FUNCTION_BLOCK "Sq_Process_IndexingUnit01"   // FB2111, GRAPH_PLUS
{ S7_Optimized_Access := 'TRUE' }
VERSION : 0.1
   VAR_INPUT
      OFF_SQ : Bool := false;   // Kette ausschalten
      INIT_SQ : Bool := false;   // Kette in Initialzustand versetzen
      ACK_EF : Bool := false;   // Alle Fehler und Störungen quittieren
      S_PREV : Bool := false;   // Vorherigen Schritt am Parameter S_NO ausgeben
      S_NEXT : Bool := false;   // Nächsten Schritt am Parameter S_NO anzeigen
      SW_AUTO : Bool := false;   // Automatischer Betrieb
      SW_TAP : Bool := false;   // Halbautomatisch/Weiterschalten mit Transition
      SW_TOP : Bool := false;   // Halbautomatisch/Ignoriere Transition
      SW_MAN : Bool := false;   // Handbetrieb
      S_SEL : Int := 0;   // Schritt auswählen, der an S_NO ausgegeben werden soll
      S_ON : Bool := false;   // Schritt aktivieren, der an Parameter S_NO anliegt
      S_OFF : Bool := false;   // Schritt deaktivieren, der an Parameter S_NO anliegt
      T_PUSH : Bool := false;   // Schaltfreigabe für Transition im halbautomatischen Betrieb
      ixStart : Bool := true;   // Startfreigabe
      ixCarrierPresent : Bool;   // WT auf dem Indexer vorhanden
      ixCheckTargetReached : Bool := false;   // 0 = Keine Sensor-Zielüberwachung nach Lift vorhanden
      ixTargetReached : Bool := false;   // WT-Sensor des nächsten Ziels
      ixReleaseHoming : Bool;   // Freigabe Grundstellungsfahrt
      ixReleaseTransfer : Bool := true;   // Freigabe der nächsten Position um WT weiterzutakten
      itCarrierReactionDelay : Time := T#350ms;   // Verzögerungszeit für die WT-Erkennung
      itMaxRuntime : Time := t#10s;   // Maximale Laufzeit für diesen Prozess
   END_VAR
   VAR_OUTPUT
      S_NO : Int := 0;   // Schrittnummer
      S_MORE : Bool := false;   // Weitere Schritte sind vorhanden und können in S_NO angezeigt werden.
      S_ACTIVE : Bool := false;   // Schritt, der an Parameter S_NO angezeigt wird, ist aktiv
      ERR_FLT : Bool := false;   // Sammelfehler Interlock oder Supervision
      AUTO_ON : Bool := false;   // Automatischer Betrieb eingeschaltet
      TAP_ON : Bool := false;   // Halbautomatischer Betrieb/Schritt mit Transition eingeschaltet
      TOP_ON : Bool := false;   // Halbautomatischer Betrieb/Ignoriere Transition eingeschaltet
      MAN_ON : Bool := false;   // Handbetrieb eingeschaltet
      qxIsActive : Bool;   // Schrittkette läuft
      qxIsInHome : Bool;   // steht in Grundstellung
      qxCarrierIsDone : Bool;   // WT-Träger ist fertig bearbeitet worden
   END_VAR
   VAR_IN_OUT
      signals : "typeStationSignals";   // Stationssteuersignale
      sq : "typeStepSequence";   // Schrittkettensteuersignale
      cylinder_lift : "typeActor_2Out2In";   // Aktor des Heber
      cylinder_stopper : "typeActor_1Out1In";   // Aktor für den Stopper
      releaseWorkStep : Bool;   // Freigabe für den externen Arbeitsschritt (muss extern zurückgesetzt werden)
   END_VAR
   VAR
      sstReleaseCycle : Struct
         ErrorAck : Bool;
         No_LastCycle : Int;
         T : Time;   // Aktive Zeit des ReleaseCycle
         Tck : Time;
         TckPrev : Time;
      END_STRUCT;
      sinstCarrierOnIndexer : TON_TIME;
      sinstCarrierLeftIndexer : TON_TIME;
      HMI_INFO : Array[0..8] of UInt;
      IF_PAR : G7_IfParPlus_V6;
      RT_DATA : G7_RTDataPlus_V6;   // Interner Datenbereich
      Automatikablauf : G7_TransitionPlus_V6;   // Transitionsstruktur
      Freigabe : G7_TransitionPlus_V6;   // Transitionsstruktur
      Trans3 : G7_TransitionPlus_V6;   // Transitionsstruktur
      Fertig : G7_TransitionPlus_V6;   // Transitionsstruktur
      Grundstellungsfahrt : G7_TransitionPlus_V6;   // Transitionsstruktur
      GST_Aktiv : G7_TransitionPlus_V6;   // Transitionsstruktur
      GST_Beendet : G7_TransitionPlus_V6;   // Transitionsstruktur
      Beendet : G7_TransitionPlus_V6;   // Transitionsstruktur
      TargetIsReached : G7_TransitionPlus_V6;   // Transitionsstruktur / Transition structure
      "Lift steht in Grundstellung_1" : G7_TransitionPlus_V6;   // Transitionsstruktur / Transition structure
      "Lift steht in Arbeitsstellung_1" : G7_TransitionPlus_V6;   // Transitionsstruktur / Transition structure
      "Lift steht in Arbeitsstellung_2" : G7_TransitionPlus_V6;   // Transitionsstruktur / Transition structure
      "WT hat Stopper verlassen" : G7_TransitionPlus_V6;   // Transitionsstruktur / Transition structure
      CarrierIsNotDone : G7_TransitionPlus_V6;   // Transitionsstruktur / Transition structure
      CarrierIsDone : G7_TransitionPlus_V6;   // Transitionsstruktur / Transition structure
      WorkstepDone : G7_TransitionPlus_V6;   // Transitionsstruktur / Transition structure
      NotDone : G7_TransitionPlus_V6;   // Transitionsstruktur / Transition structure
      WorkstepIsReleased : G7_TransitionPlus_V6;   // Transitionsstruktur / Transition structure
      EndzielFrei : G7_TransitionPlus_V6;   // Transitionsstruktur / Transition structure
      EndzielNichtFrei : G7_TransitionPlus_V6;   // Transitionsstruktur / Transition structure
      JogT2 : G7_TransitionPlus_V6;   // Transitionsstruktur / Transition structure
      JogT4 : G7_TransitionPlus_V6;   // Transitionsstruktur / Transition structure
      JogT1 : G7_TransitionPlus_V6;   // Transitionsstruktur / Transition structure
      GatesClosed : G7_TransitionPlus_V6;   // Transitionsstruktur / Transition structure
      GatesOpened : G7_TransitionPlus_V6;   // Transitionsstruktur / Transition structure
      JogT3 : G7_TransitionPlus_V6;   // Transitionsstruktur / Transition structure
      GS_GatesOpened : G7_TransitionPlus_V6;   // Transitionsstruktur / Transition structure
      Initialschritt : G7_StepPlus_V6;   // Schrittstruktur
      Grundstellung : G7_StepPlus_V6;   // Schrittstruktur
      SK_läuft : G7_StepPlus_V6;   // Schrittstruktur
      Fertigmeldung : G7_StepPlus_V6;   // Schrittstruktur
      "Start Grundstellungsfahrt" : G7_StepPlus_V6;   // Schrittstruktur
      "Fertig Grundstellungsfahrt" : G7_StepPlus_V6;   // Schrittstruktur
      Ende : G7_StepPlus_V6;   // Schrittstruktur
      WaitForTarget : G7_StepPlus_V6;   // Schrittstruktur / Step structure
      GS_CylHome : G7_StepPlus_V6;   // Schrittstruktur / Step structure
      IndexerWorkPos : G7_StepPlus_V6;   // Schrittstruktur / Step structure
      IndexerHomePos : G7_StepPlus_V6;   // Schrittstruktur / Step structure
      OpenStopper : G7_StepPlus_V6;   // Schrittstruktur / Step structure
      Decision : G7_StepPlus_V6;   // Schrittstruktur / Step structure
      CheckWorkstepDone : G7_StepPlus_V6;   // Schrittstruktur / Step structure
      Release : G7_StepPlus_V6;   // Schrittstruktur / Step structure
      Warte_Endziel_frei : G7_StepPlus_V6;   // Schrittstruktur / Step structure
      JogS2 : G7_StepPlus_V6;   // Schrittstruktur / Step structure
      JogS4 : G7_StepPlus_V6;   // Schrittstruktur / Step structure
      JogS1 : G7_StepPlus_V6;   // Schrittstruktur / Step structure
      CloseGates : G7_StepPlus_V6;   // Schrittstruktur / Step structure
      OpenGates : G7_StepPlus_V6;   // Schrittstruktur / Step structure
      JogS3 : G7_StepPlus_V6;   // Schrittstruktur / Step structure
      GS_OpenGates : G7_StepPlus_V6;   // Schrittstruktur / Step structure
      SINI : Array[0..1] of USInt;
      LSTT : Array[0..26] of USInt;
      ATAJ : Array[0..26] of USInt;
      ATAB : Array[0..26] of USInt;
      PSTT : Array[0..26] of USInt;
      NSTT : Array[0..26] of USInt;
      ASSJ : Array[0..22] of USInt;
      ASSB : Array[0..22] of USInt;
      PTTS : Array[0..22] of USInt;
      NTTS : Array[0..22] of USInt;
      SW_SQTS : Array[0..22] of USInt;
      SWITCH : Array[0..7] of USInt;
      TVX : Array[0..9] of USInt;
      TTX : Array[0..9] of USInt;
      TSX : Array[0..1] of USInt;
      S00X : Array[0..1] of USInt;
      SOFFX : Array[0..1] of USInt;
      SONX : Array[0..1] of USInt;
      SAX : Array[0..1] of USInt;
      SERRX : Array[0..23] of USInt;
      SMX : Array[0..23] of USInt;
      S0X : Array[0..23] of USInt;
      S1X : Array[0..23] of USInt;
      IL_ALARM_INST : Diag_Alarm;
      SUP_ALARM_INST : Diag_Alarm;
      STEP_TIME_ALARM_INST : Diag_Alarm;
      IEC_TIMER_INST : IEC_TIMER;
      TRANSACTION_FLAG : Bool := false;
   END_VAR
   VAR_TEMP
      txStartCondition : Bool;
      tdTckDiff : DInt;
      txCheckWorkStep : Bool;
   END_VAR
   VAR_TEMP   // added for the SCL form of the ladder/FBD networks
      _w1 : Bool;
      _w2 : Bool;
   END_VAR
   // SINI[0] := 2;
   // LSTT[0] := 255;
   // LSTT[1] := 255;
   // LSTT[2] := 255;
   // LSTT[3] := 255;
   // LSTT[4] := 255;
   // LSTT[5] := 255;
   // LSTT[6] := 255;
   // LSTT[7] := 1;
   // ATAJ[1] := 1;
   // ATAJ[2] := 2;
   // ATAJ[3] := 6;
   // ATAJ[4] := 4;
   // ATAJ[5] := 5;
   // ATAJ[6] := 3;
   // ATAJ[7] := 7;
   // ATAB[0] := 4;
   // ATAB[1] := 1;
   // ATAB[2] := 2;
   // ATAB[3] := 3;
   // ATAB[5] := 5;
   // ATAB[6] := 6;
   // ATAB[7] := 7;
   // PSTT[1] := 1;
   // PSTT[2] := 2;
   // PSTT[3] := 3;
   // PSTT[5] := 4;
   // PSTT[6] := 5;
   // PSTT[7] := 6;
   // NSTT[0] := 1;
   // NSTT[1] := 2;
   // NSTT[2] := 12;
   // NSTT[3] := 6;
   // NSTT[4] := 4;
   // NSTT[5] := 8;
   // NSTT[6] := 6;
   // NSTT[7] := 1;
   // ASSJ[1] := 1;
   // ASSJ[2] := 2;
   // ASSJ[3] := 3;
   // ASSJ[4] := 4;
   // ASSJ[5] := 5;
   // ASSJ[6] := 6;
   // ASSB[1] := 1;
   // ASSB[2] := 2;
   // ASSB[3] := 3;
   // ASSB[4] := 4;
   // ASSB[5] := 5;
   // ASSB[6] := 6;
   // PTTS[0] := 255;
   // PTTS[2] := 1;
   // PTTS[3] := 8;
   // PTTS[4] := 4;
   // PTTS[5] := 26;
   // PTTS[6] := 3;
   // NTTS[1] := 1;
   // NTTS[2] := 2;
   // NTTS[3] := 3;
   // NTTS[4] := 5;
   // NTTS[5] := 6;
   // NTTS[6] := 7;
   // SW_SQTS[1] := 1;
   // SW_SQTS[2] := 1;
   // SW_SQTS[3] := 2;
   // SW_SQTS[4] := 3;
   // SW_SQTS[5] := 3;
   // SW_SQTS[6] := 4;
   // TVX[0] := 16#1;
   // TTX[0] := 16#1;
   // TSX[0] := 16#1;
   // S00X[0] := 16#1;
   // SOFFX[0] := 16#1;
   // SONX[0] := 16#1;
   // SAX[0] := 16#1;
   // SERRX[0] := 16#1;
   // SMX[0] := 16#1;
   // S0X[0] := 16#1;
   // S1X[0] := 16#1;
   // LSTT[8] := 255;
   // ATAJ[8] := 8;
   // ATAB[8] := 8;
   // PSTT[8] := 7;
   // NSTT[8] := 3;
   // ASSJ[7] := 7;
   // ASSB[7] := 7;
   // PTTS[7] := 12;
   // NTTS[7] := 8;
   // SW_SQTS[7] := 2;
   // LSTT[9] := 255;
   // LSTT[10] := 255;
   // LSTT[11] := 255;
   // ATAJ[9] := 9;
   // ATAJ[10] := 10;
   // ATAJ[11] := 14;
   // ATAB[9] := 9;
   // ATAB[10] := 10;
   // ATAB[11] := 11;
   // PSTT[9] := 8;
   // PSTT[10] := 9;
   // PSTT[11] := 10;
   // NSTT[9] := 22;
   // NSTT[10] := 18;
   // NSTT[11] := 17;
   // ASSJ[8] := 8;
   // ASSJ[9] := 9;
   // ASSJ[10] := 10;
   // ASSB[8] := 8;
   // ASSB[9] := 9;
   // ASSB[10] := 10;
   // PTTS[8] := 5;
   // PTTS[9] := 13;
   // PTTS[10] := 25;
   // NTTS[8] := 9;
   // NTTS[9] := 10;
   // NTTS[10] := 11;
   // SW_SQTS[8] := 3;
   // SW_SQTS[9] := 5;
   // SW_SQTS[10] := 6;
   // LSTT[12] := 255;
   // LSTT[13] := 255;
   // ATAJ[12] := 12;
   // ATAJ[13] := 13;
   // ATAB[12] := 12;
   // ATAB[13] := 14;
   // PSTT[12] := 11;
   // PSTT[13] := 12;
   // NSTT[12] := 7;
   // NSTT[13] := 9;
   // ASSJ[11] := 11;
   // ASSJ[12] := 12;
   // ASSB[11] := 11;
   // ASSB[12] := 12;
   // PTTS[11] := 18;
   // PTTS[12] := 2;
   // NTTS[11] := 12;
   // NTTS[12] := 13;
   // SW_SQTS[11] := 2;
   // SW_SQTS[12] := 1;
   // LSTT[14] := 255;
   // LSTT[15] := 255;
   // ATAJ[14] := 11;
   // ATAJ[15] := 15;
   // ATAB[14] := 13;
   // ATAB[15] := 16;
   // PSTT[14] := 12;
   // PSTT[15] := 13;
   // NSTT[14] := 17;
   // NSTT[15] := 20;
   // ASSJ[13] := 13;
   // ASSJ[14] := 14;
   // ASSB[13] := 13;
   // ASSB[14] := 14;
   // PTTS[13] := 20;
   // PTTS[14] := 23;
   // NTTS[13] := 15;
   // NTTS[14] := 17;
   // SW_SQTS[13] := 5;
   // SW_SQTS[14] := 5;
   // LSTT[16] := 16;
   // ATAJ[16] := 16;
   // ATAB[16] := 15;
   // PSTT[16] := 13;
   // NSTT[16] := 16;
   // LSTT[17] := 255;
   // LSTT[18] := 255;
   // ATAJ[17] := 17;
   // ATAJ[18] := 18;
   // ATAB[17] := 17;
   // ATAB[18] := 19;
   // PSTT[17] := 14;
   // PSTT[18] := 15;
   // NSTT[17] := 16;
   // NSTT[18] := 11;
   // ASSJ[15] := 15;
   // ASSB[15] := 15;
   // PTTS[15] := 21;
   // NTTS[15] := 18;
   // SW_SQTS[15] := 7;
   // LSTT[19] := 17;
   // ATAJ[19] := 19;
   // ATAB[19] := 18;
   // PSTT[19] := 15;
   // NSTT[19] := 17;
   // ASSJ[16] := 16;
   // ASSB[16] := 16;
   // PTTS[16] := 17;
   // NTTS[16] := 20;
   // SW_SQTS[16] := 5;
   // LSTT[20] := 255;
   // LSTT[21] := 255;
   // LSTT[22] := 255;
   // LSTT[23] := 255;
   // LSTT[24] := 255;
   // LSTT[25] := 255;
   // ATAJ[20] := 20;
   // ATAJ[21] := 21;
   // ATAJ[22] := 22;
   // ATAJ[23] := 23;
   // ATAJ[24] := 24;
   // ATAJ[25] := 25;
   // ATAB[20] := 20;
   // ATAB[21] := 21;
   // ATAB[22] := 22;
   // ATAB[23] := 23;
   // ATAB[24] := 24;
   // ATAB[25] := 25;
   // PSTT[20] := 16;
   // PSTT[21] := 17;
   // PSTT[22] := 18;
   // PSTT[23] := 19;
   // PSTT[24] := 20;
   // PSTT[25] := 21;
   // NSTT[20] := 13;
   // NSTT[21] := 15;
   // NSTT[22] := 19;
   // NSTT[23] := 14;
   // NSTT[24] := 21;
   // NSTT[25] := 10;
   // ASSJ[17] := 17;
   // ASSJ[18] := 18;
   // ASSJ[19] := 19;
   // ASSJ[20] := 20;
   // ASSJ[21] := 21;
   // ASSB[17] := 17;
   // ASSB[18] := 18;
   // ASSB[19] := 19;
   // ASSB[20] := 20;
   // ASSB[21] := 21;
   // PTTS[17] := 11;
   // PTTS[18] := 10;
   // PTTS[19] := 22;
   // PTTS[20] := 15;
   // PTTS[21] := 24;
   // NTTS[17] := 21;
   // NTTS[18] := 22;
   // NTTS[19] := 23;
   // NTTS[20] := 24;
   // NTTS[21] := 25;
   // SW_SQTS[17] := 7;
   // SW_SQTS[18] := 5;
   // SW_SQTS[19] := 5;
   // SW_SQTS[20] := 6;
   // SW_SQTS[21] := 6;
   // LSTT[26] := 255;
   // ATAJ[26] := 26;
   // ATAB[26] := 26;
   // PSTT[26] := 22;
   // NSTT[26] := 5;
   // ASSJ[22] := 22;
   // ASSB[22] := 22;
   // PTTS[22] := 9;
   // NTTS[22] := 26;
   // SW_SQTS[22] := 3;
BEGIN
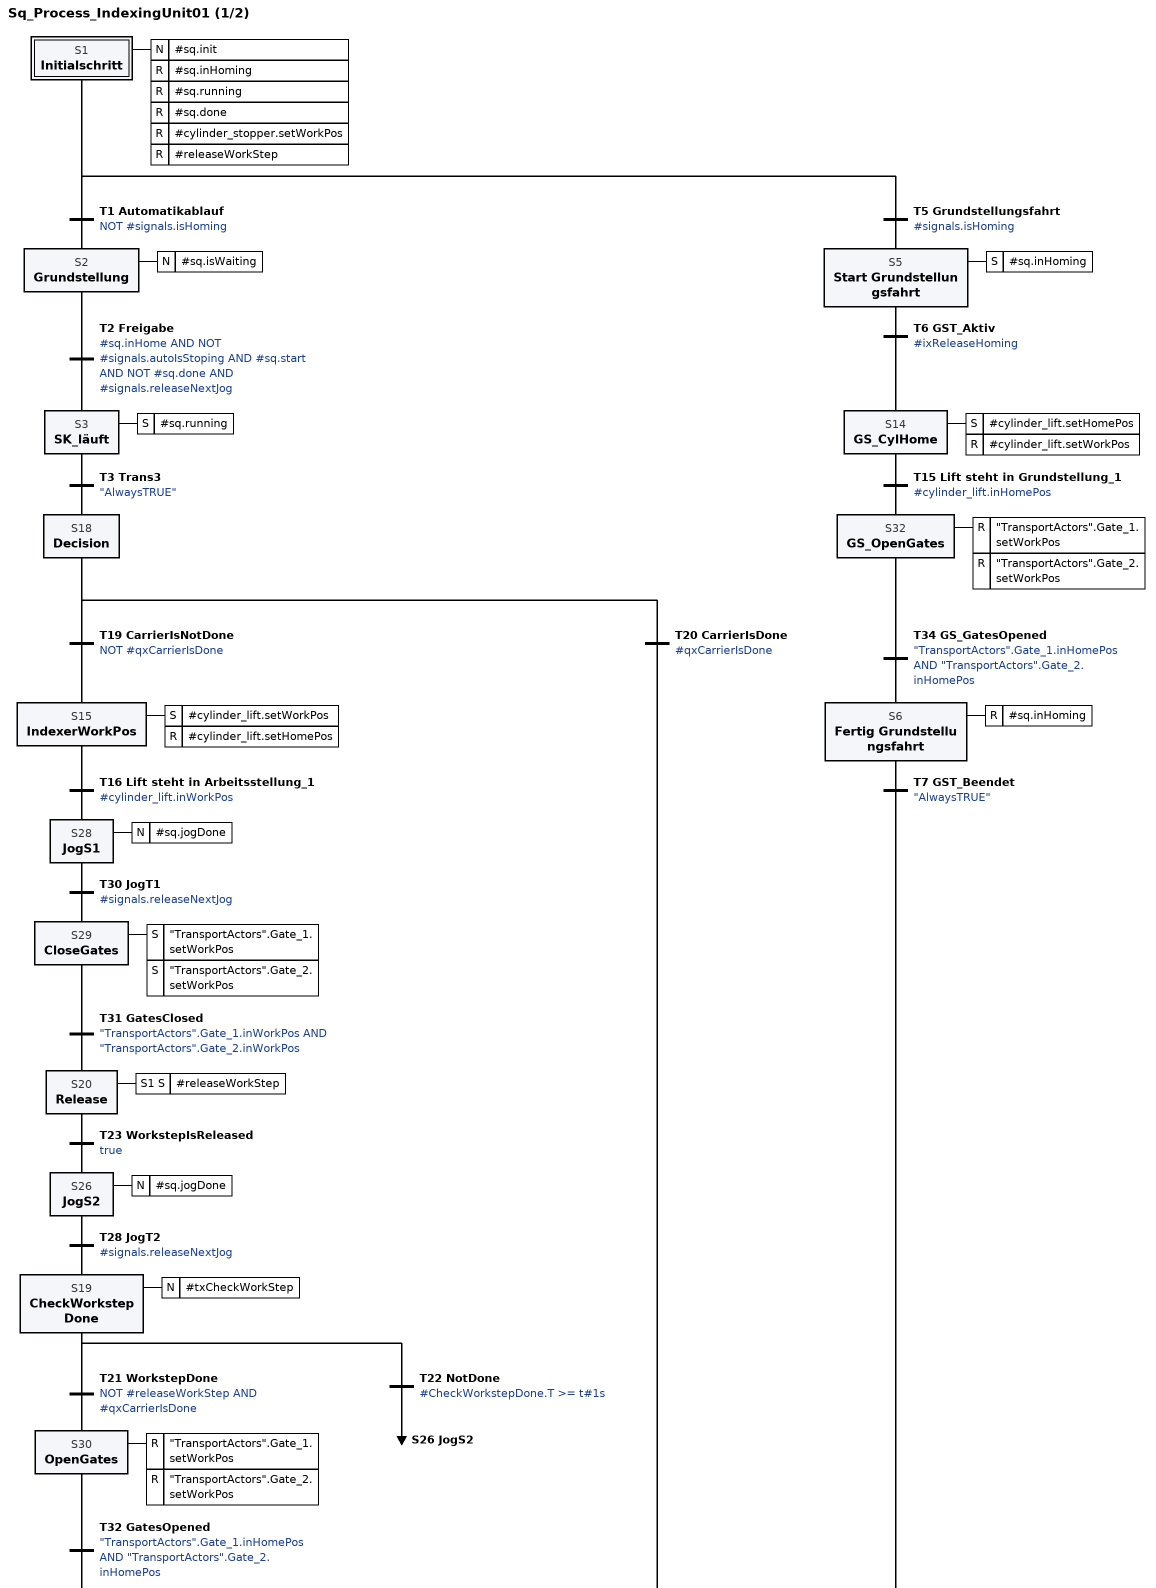
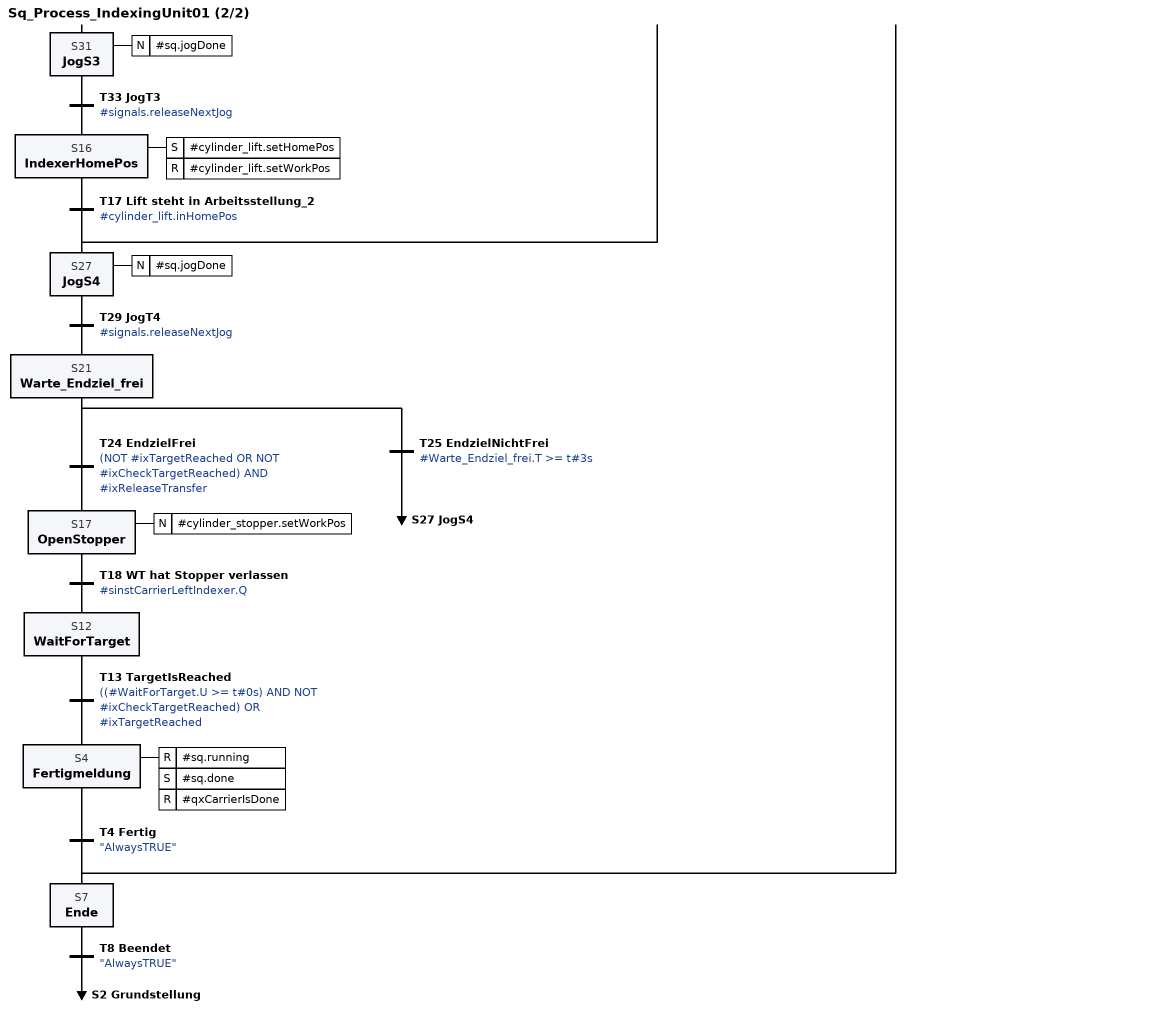
   // permanent pre-instructions
   NETWORK 1
   TITLE = Schrittkette verfügbar
      #sq.exists := true;
   NETWORK 2
   TITLE = WT auf dem Indexer
      #sinstCarrierOnIndexer(IN := #ixCarrierPresent, PT := #itCarrierReactionDelay);   // TON
   NETWORK 3
   TITLE = WT hat den Indexer verlassen
      #sinstCarrierLeftIndexer(IN := NOT #ixCarrierPresent, PT := #itCarrierReactionDelay);   // TON
   NETWORK 4
   TITLE = Schrittkette in Grundstellung (Erweitern)
      #sq.inHome := #Grundstellung.X AND #cylinder_lift.inHomePos AND #cylinder_stopper.inHomePos AND "TransportActors".Gate_1.inHomePos AND "TransportActors".Gate_2.inHomePos;
   NETWORK 5
   TITLE = Startbedingung (Erweitern)
      #txStartCondition := #ixStart AND #sinstCarrierOnIndexer.Q;
   NETWORK 6
   TITLE = Schrittkette starten
      #sq.start := #sq.inHome AND NOT #sq.running AND #signals.releaseCycle AND NOT #signals.isHoming AND #txStartCondition;
      IF #sq.start THEN #sq.done := FALSE; END_IF;
   NETWORK 7
   TITLE = ReleaseCycle Timer
      // ENO of a box is taken as its EN; it also drops when the box reports an error
      #_w1 := #ERR_FLT AND #ACK_EF;
      #_w2 := #_w1 AND NOT #sstReleaseCycle.ErrorAck;   // rising edge
      #sstReleaseCycle.ErrorAck := #_w1;
      IF (#S_NO <> #sstReleaseCycle.No_LastCycle) OR #_w2 THEN
          #sstReleaseCycle.T := T#0MS;
          #sstReleaseCycle.TckPrev := #sstReleaseCycle.Tck;
          #sstReleaseCycle.No_LastCycle := #S_NO;
      END_IF;
      #sstReleaseCycle.Tck := TIME_TCK();
      #tdTckDiff := #sstReleaseCycle.Tck - #sstReleaseCycle.TckPrev;
      #sstReleaseCycle.TckPrev := #sstReleaseCycle.Tck;
      IF (0 <= #tdTckDiff) AND (#tdTckDiff <= 1000) AND #signals.releaseCycle THEN
          #sstReleaseCycle.T := #sstReleaseCycle.T + #tdTckDiff;
      END_IF;

   // sequencer 1
   INITIAL_STEP Initialschritt:   // S1, max time T#10S, warning time T#7S
              N    #sq.init
              R    #sq.inHoming
              R    #sq.running
              R    #sq.done
              R    #cylinder_stopper.setWorkPos
              R    #releaseWorkStep
   END_STEP
   TRANSITION Automatikablauf FROM Initialschritt TO Grundstellung   // T1
      := NOT #signals.isHoming;
   END_TRANSITION
   TRANSITION Grundstellungsfahrt FROM Initialschritt TO "Start Grundstellungsfahrt"   // T5
      := #signals.isHoming;
   END_TRANSITION
   STEP Grundstellung:   // S2, max time T#10S, warning time T#7S
              N    #sq.isWaiting
   END_STEP
   TRANSITION Freigabe FROM Grundstellung TO SK_läuft   // T2
      := #sq.inHome AND NOT #signals.autoIsStoping AND #sq.start AND NOT #sq.done AND #signals.releaseNextJog;
   END_TRANSITION
   STEP SK_läuft:   // S3, max time T#10S, warning time T#7S
              S    #sq.running
   END_STEP
   TRANSITION Trans3 FROM SK_läuft TO Decision   // T3
      := "AlwaysTRUE";
   END_TRANSITION
   STEP Fertigmeldung:   // S4, max time T#10S, warning time T#7S
              R    #sq.running
              S    #sq.done
              R    #qxCarrierIsDone
   END_STEP
   TRANSITION Fertig FROM Fertigmeldung TO Ende   // T4
      := "AlwaysTRUE";
   END_TRANSITION
   STEP "Start Grundstellungsfahrt":   // S5, max time T#10S, warning time T#7S
              S    #sq.inHoming
   END_STEP
   TRANSITION GST_Aktiv FROM "Start Grundstellungsfahrt" TO GS_CylHome   // T6
      := #ixReleaseHoming;
   END_TRANSITION
   STEP "Fertig Grundstellungsfahrt":   // S6, max time T#10S, warning time T#7S
              R    #sq.inHoming
   END_STEP
   TRANSITION GST_Beendet FROM "Fertig Grundstellungsfahrt" TO Ende   // T7
      := "AlwaysTRUE";
   END_TRANSITION
   STEP Ende:   // S7, max time T#10S, warning time T#7S
   END_STEP
   TRANSITION Beendet FROM Ende TO Grundstellung   // T8, jump
      := "AlwaysTRUE";
   END_TRANSITION
   STEP JogS2:   // S26, max time T#10S, warning time T#7S
              N    #sq.jogDone
   END_STEP
   TRANSITION JogT2 FROM JogS2 TO CheckWorkstepDone   // T28
      := #signals.releaseNextJog;
   END_TRANSITION
   STEP IndexerHomePos:   // S16, max time T#10S, warning time T#7S
      supervision V := #IndexerHomePos.X AND #cylinder_lift.inError;
              S    #cylinder_lift.setHomePos
              R    #cylinder_lift.setWorkPos
   END_STEP
   TRANSITION "Lift steht in Arbeitsstellung_2" FROM IndexerHomePos TO JogS4   // T17
      := #cylinder_lift.inHomePos;
   END_TRANSITION
   STEP OpenStopper:   // S17, max time T#10S, warning time T#7S
      supervision V := #OpenStopper.X AND #cylinder_stopper.inError;
              N    #cylinder_stopper.setWorkPos
   END_STEP
   TRANSITION "WT hat Stopper verlassen" FROM OpenStopper TO WaitForTarget   // T18
      := #sinstCarrierLeftIndexer.Q;
   END_TRANSITION
   STEP JogS4:   // S27, max time T#10S, warning time T#7S
              N    #sq.jogDone
   END_STEP
   TRANSITION JogT4 FROM JogS4 TO Warte_Endziel_frei   // T29
      := #signals.releaseNextJog;
   END_TRANSITION
   STEP WaitForTarget:   // S12, max time T#10S, warning time T#7S
      supervision V := #sstReleaseCycle.T >= #itMaxRuntime;
   END_STEP
   TRANSITION TargetIsReached FROM WaitForTarget TO Fertigmeldung   // T13
      := ((#WaitForTarget.U >= t#0s) AND NOT #ixCheckTargetReached) OR #ixTargetReached;
   END_TRANSITION
   STEP Decision:   // S18, max time T#10S, warning time T#7S
   END_STEP
   TRANSITION CarrierIsNotDone FROM Decision TO IndexerWorkPos   // T19
      := NOT #qxCarrierIsDone;
   END_TRANSITION
   TRANSITION CarrierIsDone FROM Decision TO JogS4   // T20
      := #qxCarrierIsDone;
   END_TRANSITION
   STEP GS_CylHome:   // S14, max time T#10S, warning time T#7S
      supervision V := #GS_CylHome.X AND #cylinder_lift.inError;
              S    #cylinder_lift.setHomePos
              R    #cylinder_lift.setWorkPos
   END_STEP
   TRANSITION "Lift steht in Grundstellung_1" FROM GS_CylHome TO GS_OpenGates   // T15
      := #cylinder_lift.inHomePos;
   END_TRANSITION
   STEP IndexerWorkPos:   // S15, max time T#10S, warning time T#7S
      supervision V := #IndexerWorkPos.X AND #cylinder_lift.inError;
              S    #cylinder_lift.setWorkPos
              R    #cylinder_lift.setHomePos
   END_STEP
   TRANSITION "Lift steht in Arbeitsstellung_1" FROM IndexerWorkPos TO JogS1   // T16
      := #cylinder_lift.inWorkPos;
   END_TRANSITION
   STEP CheckWorkstepDone:   // S19, max time T#10S, warning time T#7S
              N    #txCheckWorkStep
   END_STEP
   TRANSITION WorkstepDone FROM CheckWorkstepDone TO OpenGates   // T21
      := NOT #releaseWorkStep AND #qxCarrierIsDone;
   END_TRANSITION
   TRANSITION NotDone FROM CheckWorkstepDone TO JogS2   // T22, jump
      := #CheckWorkstepDone.T >= t#1s;
   END_TRANSITION
   STEP Release:   // S20, max time T#10S, warning time T#7S
          S1  S    #releaseWorkStep
   END_STEP
   TRANSITION WorkstepIsReleased FROM Release TO JogS2   // T23
      := true;
   END_TRANSITION
   STEP Warte_Endziel_frei:   // S21, max time T#10S, warning time T#7S
   END_STEP
   TRANSITION EndzielFrei FROM Warte_Endziel_frei TO OpenStopper   // T24
      := (NOT #ixTargetReached OR NOT #ixCheckTargetReached) AND #ixReleaseTransfer;
   END_TRANSITION
   TRANSITION EndzielNichtFrei FROM Warte_Endziel_frei TO JogS4   // T25, jump
      := #Warte_Endziel_frei.T >= t#3s;
   END_TRANSITION
   STEP JogS1:   // S28, max time T#10S, warning time T#7S
              N    #sq.jogDone
   END_STEP
   TRANSITION JogT1 FROM JogS1 TO CloseGates   // T30
      := #signals.releaseNextJog;
   END_TRANSITION
   STEP CloseGates:   // S29, max time T#10S, warning time T#7S
      supervision V := (#sstReleaseCycle.T >= #itMaxRuntime) OR (("TransportActors".Gate_1.inError OR "TransportActors".Gate_2.inError) AND #CloseGates.X);
              S    "TransportActors".Gate_1.setWorkPos
              S    "TransportActors".Gate_2.setWorkPos
   END_STEP
   TRANSITION GatesClosed FROM CloseGates TO Release   // T31
      := "TransportActors".Gate_1.inWorkPos AND "TransportActors".Gate_2.inWorkPos;
   END_TRANSITION
   STEP OpenGates:   // S30, max time T#10S, warning time T#7S
      supervision V := (#sstReleaseCycle.T >= #itMaxRuntime) OR (("TransportActors".Gate_1.inError OR "TransportActors".Gate_2.inError) AND #OpenGates.X);
              R    "TransportActors".Gate_1.setWorkPos
              R    "TransportActors".Gate_2.setWorkPos
   END_STEP
   TRANSITION GatesOpened FROM OpenGates TO JogS3   // T32
      := "TransportActors".Gate_1.inHomePos AND "TransportActors".Gate_2.inHomePos;
   END_TRANSITION
   STEP JogS3:   // S31, max time T#10S, warning time T#7S
              N    #sq.jogDone
   END_STEP
   TRANSITION JogT3 FROM JogS3 TO IndexerHomePos   // T33
      := #signals.releaseNextJog;
   END_TRANSITION
   STEP GS_OpenGates:   // S32, max time T#10S, warning time T#7S
      supervision V := (#sstReleaseCycle.T >= #itMaxRuntime) OR (("TransportActors".Gate_1.inError OR "TransportActors".Gate_2.inError) AND #GS_OpenGates.X);
              R    "TransportActors".Gate_1.setWorkPos
              R    "TransportActors".Gate_2.setWorkPos
   END_STEP
   TRANSITION GS_GatesOpened FROM GS_OpenGates TO "Fertig Grundstellungsfahrt"   // T34
      := "TransportActors".Gate_1.inHomePos AND "TransportActors".Gate_2.inHomePos;
   END_TRANSITION

   // permanent post-instructions
   NETWORK 1
   TITLE = Störungssignal weitergeben
      #sq.error := #ERR_FLT;
   NETWORK 2
   TITLE = Ablauf ist aktiv
      #qxIsActive := #sq.running;
   NETWORK 3
   TITLE = steht in Grundstellung
      #qxIsInHome := #sq.inHome AND NOT #sq.running;
   NETWORK 4
   TITLE = WT-Träger ist fertig bearbeitet worden
      IF NOT #releaseWorkStep AND #txCheckWorkStep THEN #qxCarrierIsDone := TRUE; END_IF;
END_FUNCTION_BLOCK

FUNCTION "FG10StepSequences" : Void   // FC2010, FBD
TITLE = Schrittkettensteuerung
{ S7_Optimized_Access := 'TRUE' }
VERSION : 0.1
// Ersteller: Andreas Fast Automation
// E-Mail: automation@fast-andreas.de
// 
// Projekt dient zu Demonstrationszwecken und frei genutzt werden.
// 
// Bausteinbeschreibung:
   VAR_IN_OUT
      station : "typeStation";
   END_VAR
   VAR_TEMP
      tempInit : Bool;
      tempAck : Bool;
      tempSwAuto : Bool;
      tempSwMan : Bool;
      tempSwTap : Bool;
      tempPush : Bool;
   END_VAR
BEGIN

REGION Network 1: Graph Parameter
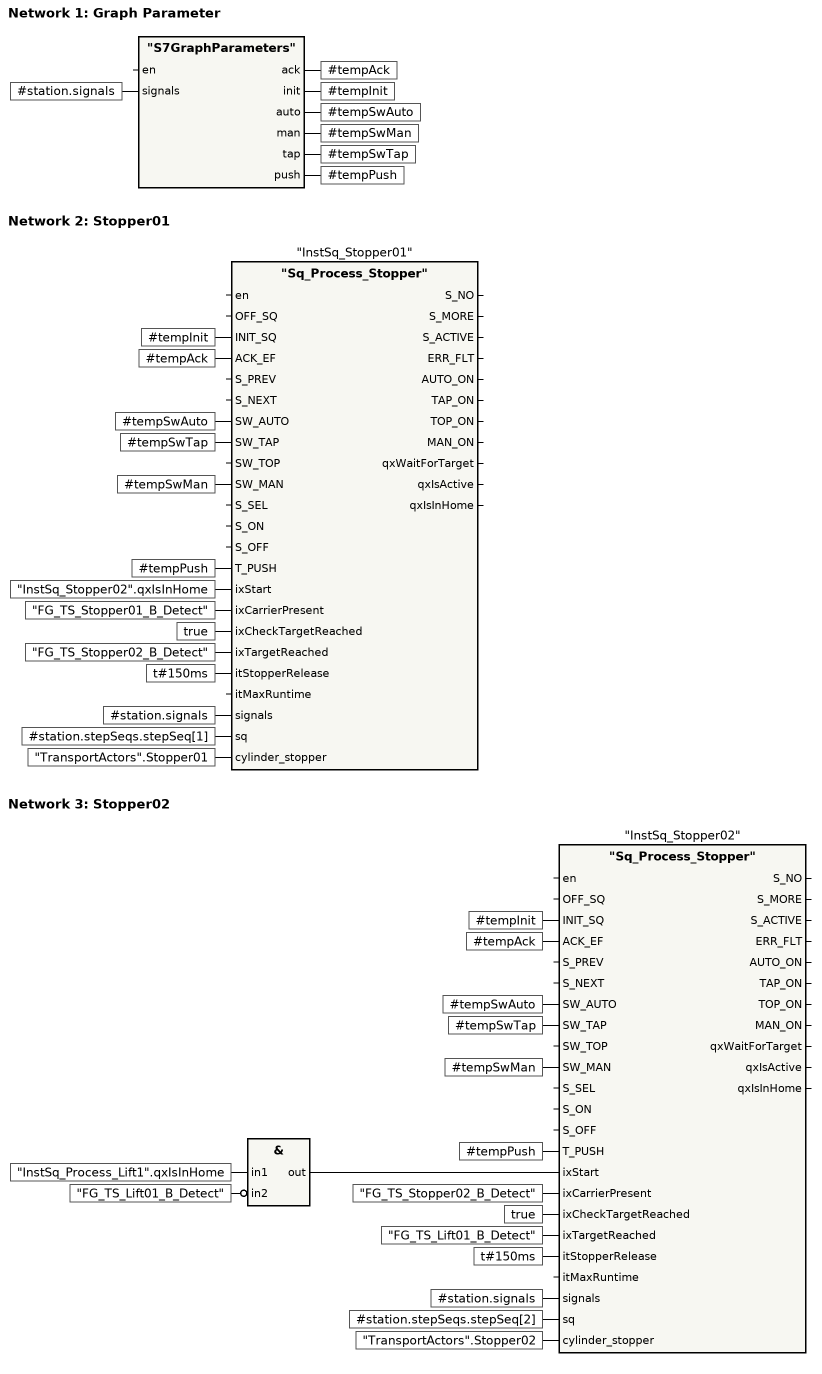
   "S7GraphParameters"(signals := #station.signals,
                       ack => #tempAck,
                       init => #tempInit,
                       auto => #tempSwAuto,
                       man => #tempSwMan,
                       tap => #tempSwTap,
                       push => #tempPush);
END_REGION

REGION Network 2: Stopper01
   "InstSq_Stopper01"(INIT_SQ := #tempInit,   // "Sq_Process_Stopper"
                      ACK_EF := #tempAck,
                      SW_AUTO := #tempSwAuto,
                      SW_TAP := #tempSwTap,
                      SW_MAN := #tempSwMan,
                      T_PUSH := #tempPush,
                      ixStart := "InstSq_Stopper02".qxIsInHome,
                      ixCarrierPresent := "FG_TS_Stopper01_B_Detect",
                      ixCheckTargetReached := true,
                      ixTargetReached := "FG_TS_Stopper02_B_Detect",
                      itStopperRelease := t#150ms,
                      signals := #station.signals,
                      sq := #station.stepSeqs.stepSeq[1],
                      cylinder_stopper := "TransportActors".Stopper01);
END_REGION

REGION Network 3: Stopper02
   "InstSq_Stopper02"(INIT_SQ := #tempInit,   // "Sq_Process_Stopper"
                      ACK_EF := #tempAck,
                      SW_AUTO := #tempSwAuto,
                      SW_TAP := #tempSwTap,
                      SW_MAN := #tempSwMan,
                      T_PUSH := #tempPush,
                      ixStart := "InstSq_Process_Lift1".qxIsInHome AND NOT "FG_TS_Lift01_B_Detect",
                      ixCarrierPresent := "FG_TS_Stopper02_B_Detect",
                      ixCheckTargetReached := true,
                      ixTargetReached := "FG_TS_Lift01_B_Detect",
                      itStopperRelease := t#150ms,
                      signals := #station.signals,
                      sq := #station.stepSeqs.stepSeq[2],
                      cylinder_stopper := "TransportActors".Stopper02);
END_REGION

REGION Network 4: Lift 1
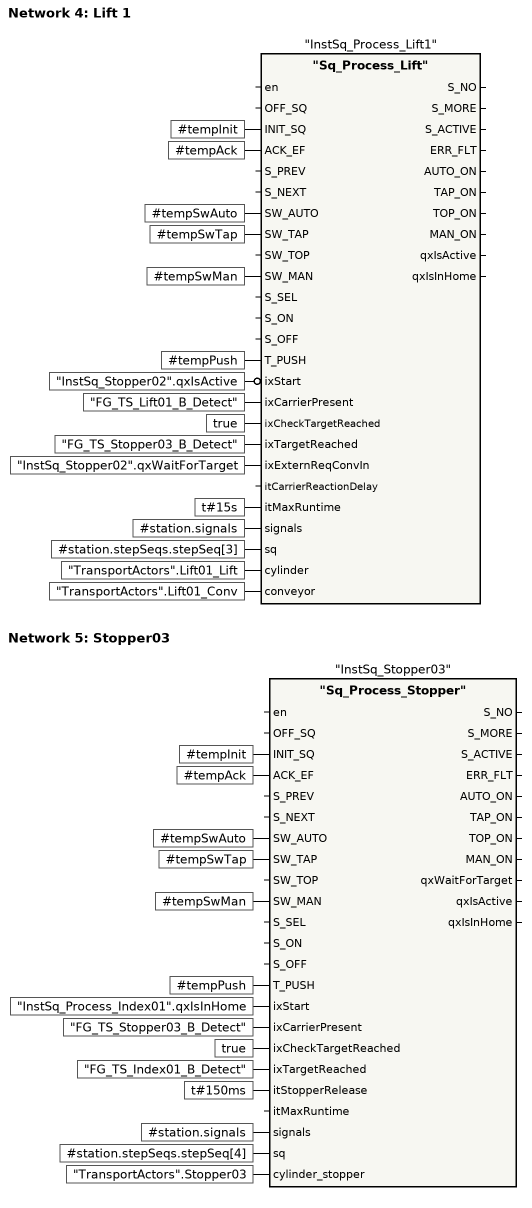
   "InstSq_Process_Lift1"(INIT_SQ := #tempInit,   // "Sq_Process_Lift"
                          ACK_EF := #tempAck,
                          SW_AUTO := #tempSwAuto,
                          SW_TAP := #tempSwTap,
                          SW_MAN := #tempSwMan,
                          T_PUSH := #tempPush,
                          ixStart := NOT "InstSq_Stopper02".qxIsActive,
                          ixCarrierPresent := "FG_TS_Lift01_B_Detect",
                          ixCheckTargetReached := true,
                          ixTargetReached := "FG_TS_Stopper03_B_Detect",
                          ixExternReqConvIn := "InstSq_Stopper02".qxWaitForTarget,
                          itMaxRuntime := t#15s,
                          signals := #station.signals,
                          sq := #station.stepSeqs.stepSeq[3],
                          cylinder := "TransportActors".Lift01_Lift,
                          conveyor := "TransportActors".Lift01_Conv);
END_REGION

REGION Network 5: Stopper03
   "InstSq_Stopper03"(INIT_SQ := #tempInit,   // "Sq_Process_Stopper"
                      ACK_EF := #tempAck,
                      SW_AUTO := #tempSwAuto,
                      SW_TAP := #tempSwTap,
                      SW_MAN := #tempSwMan,
                      T_PUSH := #tempPush,
                      ixStart := "InstSq_Process_Index01".qxIsInHome,
                      ixCarrierPresent := "FG_TS_Stopper03_B_Detect",
                      ixCheckTargetReached := true,
                      ixTargetReached := "FG_TS_Index01_B_Detect",
                      itStopperRelease := t#150ms,
                      signals := #station.signals,
                      sq := #station.stepSeqs.stepSeq[4],
                      cylinder_stopper := "TransportActors".Stopper03);
END_REGION

REGION Network 6: Index01
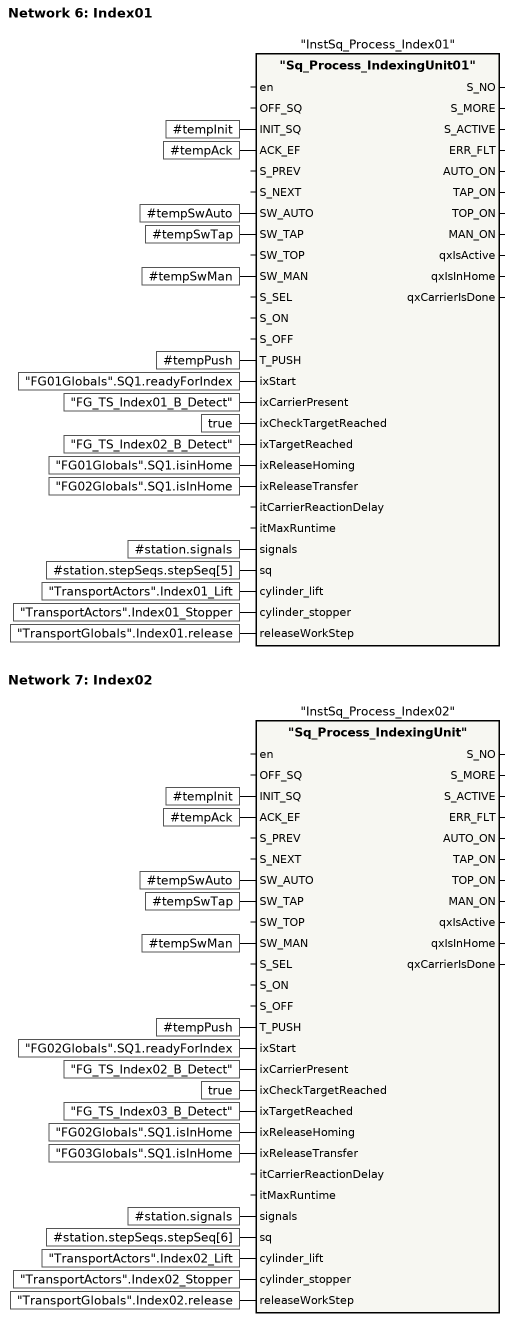
   "InstSq_Process_Index01"(INIT_SQ := #tempInit,   // "Sq_Process_IndexingUnit01"
                           ACK_EF := #tempAck,
                           SW_AUTO := #tempSwAuto,
                           SW_TAP := #tempSwTap,
                           SW_MAN := #tempSwMan,
                           T_PUSH := #tempPush,
                           ixStart := "FG01Globals".SQ1.readyForIndex,
                           ixCarrierPresent := "FG_TS_Index01_B_Detect",
                           ixCheckTargetReached := true,
                           ixTargetReached := "FG_TS_Index02_B_Detect",
                           ixReleaseHoming := "FG01Globals".SQ1.isinHome,
                           ixReleaseTransfer := "FG02Globals".SQ1.isInHome,
                           signals := #station.signals,
                           sq := #station.stepSeqs.stepSeq[5],
                           cylinder_lift := "TransportActors".Index01_Lift,
                           cylinder_stopper := "TransportActors".Index01_Stopper,
                           releaseWorkStep := "TransportGlobals".Index01.release);
END_REGION

REGION Network 7: Index02
   "InstSq_Process_Index02"(INIT_SQ := #tempInit,   // "Sq_Process_IndexingUnit"
                           ACK_EF := #tempAck,
                           SW_AUTO := #tempSwAuto,
                           SW_TAP := #tempSwTap,
                           SW_MAN := #tempSwMan,
                           T_PUSH := #tempPush,
                           ixStart := "FG02Globals".SQ1.readyForIndex,
                           ixCarrierPresent := "FG_TS_Index02_B_Detect",
                           ixCheckTargetReached := true,
                           ixTargetReached := "FG_TS_Index03_B_Detect",
                           ixReleaseHoming := "FG02Globals".SQ1.isInHome,
                           ixReleaseTransfer := "FG03Globals".SQ1.isInHome,
                           signals := #station.signals,
                           sq := #station.stepSeqs.stepSeq[6],
                           cylinder_lift := "TransportActors".Index02_Lift,
                           cylinder_stopper := "TransportActors".Index02_Stopper,
                           releaseWorkStep := "TransportGlobals".Index02.release);
END_REGION

REGION Network 8: Index03
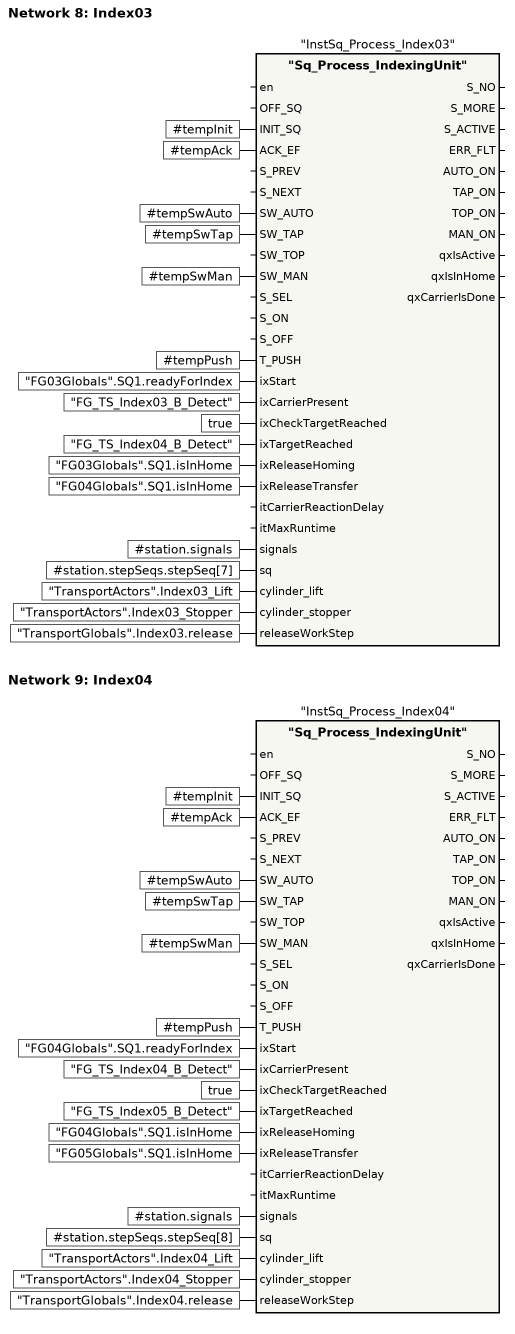
   "InstSq_Process_Index03"(INIT_SQ := #tempInit,   // "Sq_Process_IndexingUnit"
                           ACK_EF := #tempAck,
                           SW_AUTO := #tempSwAuto,
                           SW_TAP := #tempSwTap,
                           SW_MAN := #tempSwMan,
                           T_PUSH := #tempPush,
                           ixStart := "FG03Globals".SQ1.readyForIndex,
                           ixCarrierPresent := "FG_TS_Index03_B_Detect",
                           ixCheckTargetReached := true,
                           ixTargetReached := "FG_TS_Index04_B_Detect",
                           ixReleaseHoming := "FG03Globals".SQ1.isInHome,
                           ixReleaseTransfer := "FG04Globals".SQ1.isInHome,
                           signals := #station.signals,
                           sq := #station.stepSeqs.stepSeq[7],
                           cylinder_lift := "TransportActors".Index03_Lift,
                           cylinder_stopper := "TransportActors".Index03_Stopper,
                           releaseWorkStep := "TransportGlobals".Index03.release);
END_REGION

REGION Network 9: Index04
   "InstSq_Process_Index04"(INIT_SQ := #tempInit,   // "Sq_Process_IndexingUnit"
                           ACK_EF := #tempAck,
                           SW_AUTO := #tempSwAuto,
                           SW_TAP := #tempSwTap,
                           SW_MAN := #tempSwMan,
                           T_PUSH := #tempPush,
                           ixStart := "FG04Globals".SQ1.readyForIndex,
                           ixCarrierPresent := "FG_TS_Index04_B_Detect",
                           ixCheckTargetReached := true,
                           ixTargetReached := "FG_TS_Index05_B_Detect",
                           ixReleaseHoming := "FG04Globals".SQ1.isInHome,
                           ixReleaseTransfer := "FG05Globals".SQ1.isInHome,
                           signals := #station.signals,
                           sq := #station.stepSeqs.stepSeq[8],
                           cylinder_lift := "TransportActors".Index04_Lift,
                           cylinder_stopper := "TransportActors".Index04_Stopper,
                           releaseWorkStep := "TransportGlobals".Index04.release);
END_REGION

REGION Network 10: Index05
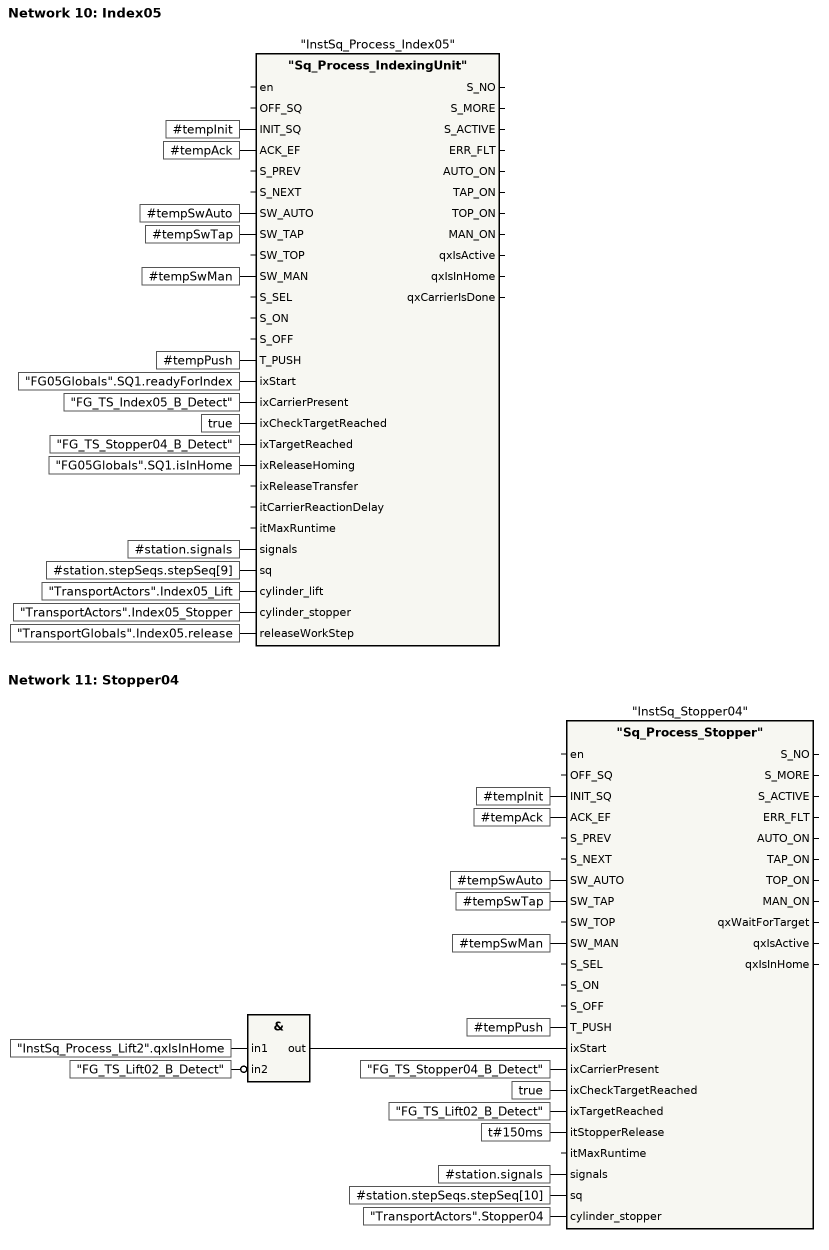
   "InstSq_Process_Index05"(INIT_SQ := #tempInit,   // "Sq_Process_IndexingUnit"
                           ACK_EF := #tempAck,
                           SW_AUTO := #tempSwAuto,
                           SW_TAP := #tempSwTap,
                           SW_MAN := #tempSwMan,
                           T_PUSH := #tempPush,
                           ixStart := "FG05Globals".SQ1.readyForIndex,
                           ixCarrierPresent := "FG_TS_Index05_B_Detect",
                           ixCheckTargetReached := true,
                           ixTargetReached := "FG_TS_Stopper04_B_Detect",
                           ixReleaseHoming := "FG05Globals".SQ1.isInHome,
                           signals := #station.signals,
                           sq := #station.stepSeqs.stepSeq[9],
                           cylinder_lift := "TransportActors".Index05_Lift,
                           cylinder_stopper := "TransportActors".Index05_Stopper,
                           releaseWorkStep := "TransportGlobals".Index05.release);
END_REGION

REGION Network 11: Stopper04
   "InstSq_Stopper04"(INIT_SQ := #tempInit,   // "Sq_Process_Stopper"
                      ACK_EF := #tempAck,
                      SW_AUTO := #tempSwAuto,
                      SW_TAP := #tempSwTap,
                      SW_MAN := #tempSwMan,
                      T_PUSH := #tempPush,
                      ixStart := "InstSq_Process_Lift2".qxIsInHome AND NOT "FG_TS_Lift02_B_Detect",
                      ixCarrierPresent := "FG_TS_Stopper04_B_Detect",
                      ixCheckTargetReached := true,
                      ixTargetReached := "FG_TS_Lift02_B_Detect",
                      itStopperRelease := t#150ms,
                      signals := #station.signals,
                      sq := #station.stepSeqs.stepSeq[10],
                      cylinder_stopper := "TransportActors".Stopper04);
END_REGION

REGION Network 12: Lift 2
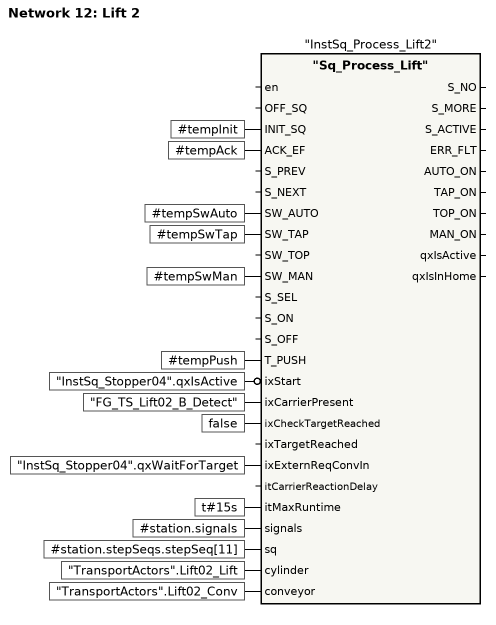
   "InstSq_Process_Lift2"(INIT_SQ := #tempInit,   // "Sq_Process_Lift"
                          ACK_EF := #tempAck,
                          SW_AUTO := #tempSwAuto,
                          SW_TAP := #tempSwTap,
                          SW_MAN := #tempSwMan,
                          T_PUSH := #tempPush,
                          ixStart := NOT "InstSq_Stopper04".qxIsActive,
                          ixCarrierPresent := "FG_TS_Lift02_B_Detect",
                          ixCheckTargetReached := false,
                          ixExternReqConvIn := "InstSq_Stopper04".qxWaitForTarget,
                          itMaxRuntime := t#15s,
                          signals := #station.signals,
                          sq := #station.stepSeqs.stepSeq[11],
                          cylinder := "TransportActors".Lift02_Lift,
                          conveyor := "TransportActors".Lift02_Conv);
END_REGION
END_FUNCTION

// folder: 9. Library

FUNCTION_BLOCK "MachineControl"   // FB9000, FBD
TITLE = Maschinensteuerung
{ S7_Optimized_Access := 'TRUE' }
VERSION : 0.1
// Ersteller: Andreas Fast Automation
// E-Mail: automation@fast-andreas.de
// 
// Projekt dient zu Demonstrationszwecken und frei genutzt werden.
// 
// Bausteinbeschreibung:
   VAR_INPUT
      firstPlcCycle : Bool;   // Erster Zyklus
      configNoControlOff : Bool := true;   // 1 = Ohne controlOff (Ein-/Ausschalten nur über controlOn)
      controlOn : Bool;   // Input 'control on' (if true)
      contolOff : Bool := true;   // Input 'control off' (if false)
      automaticMode : Bool;   // Input 'automatic/manual operation'
      singleStep : Bool;   // Input 'single step'
      autoStart : Bool;   // Input 'automatic start'
      autoStop : Bool;   // Input ' automatic stop'
      immediateStop : Bool;   // Input 'immediate stop'
      reset : Bool;   // Input 'machine reset'
      acknowledge : Bool;   // Input ' acknowledgement'
      errFlt : Bool;   // Input 'machine error'
   END_VAR
   VAR_OUTPUT
      controlOnLight : Bool;   // Steuerung Ein = Dauerlicht; Steuerung fährt hoch = Blinklicht; Steuerung aus = Licht aus
      setupOnLight : Bool;   // Einrichten aktiv = Ein
      automaticRunsLight : Bool;   // Automatik aktiv = Dauerlicht; Teilautomatik = Blinklicht; Automatik aus = Licht aus
      singleStepLight : Bool;   // Einzelschritt läuft = Dauerlicht
      automaticStopsLight : Bool;   // Automatik stoppt = Blinklicht
      errFltLight : Bool;   // Störung = Dauerlicht
      homingLight : Bool;   // Grundstellungsfahrt läuft = Blinklicht; Maschine in Grundstellung = Dauerlicht
      manAutoLight : Bool;   // Auto = Dauerlicht, Hand = Licht aus
   END_VAR
   VAR_IN_OUT
      safety : "typeMachineSafety";
      machine : "typeMachine";
      stations : "typeStations";
      manualMovement : "typeManualMovements";
      plcErrMsg : "typePlcErrMsg";
      hmiErrMsg : "typeHmiErrMsg";
   END_VAR
   VAR
      statControlRunUp : Bool;
      statTrigControlOn : Bool;
      statTrigReset : Bool;
      statTrigSingleStep : Bool;
      statTrigAutoStart : Bool;
      statTrigHomingDone : Bool;
      statFirstCycle : Bool;
      statStationsAllStopped : Bool;
      statStationsAllRunning : Bool;
      statAnyStationInAutoRun : Bool;
      instTonRunUp : TON_TIME;
      instAlarmHandler : "AlarmHandler";
   END_VAR
   VAR_TEMP
      tempStationError : Bool;
      tempStationsInSetup : Bool;
      tempAnyJogIsActive : Bool;
   END_VAR
   VAR_TEMP   // added for the SCL form of the ladder/FBD networks
      _w1 : Bool;
      _w2 : Bool;
   END_VAR
BEGIN

REGION Network 1: Meldungen auslösen
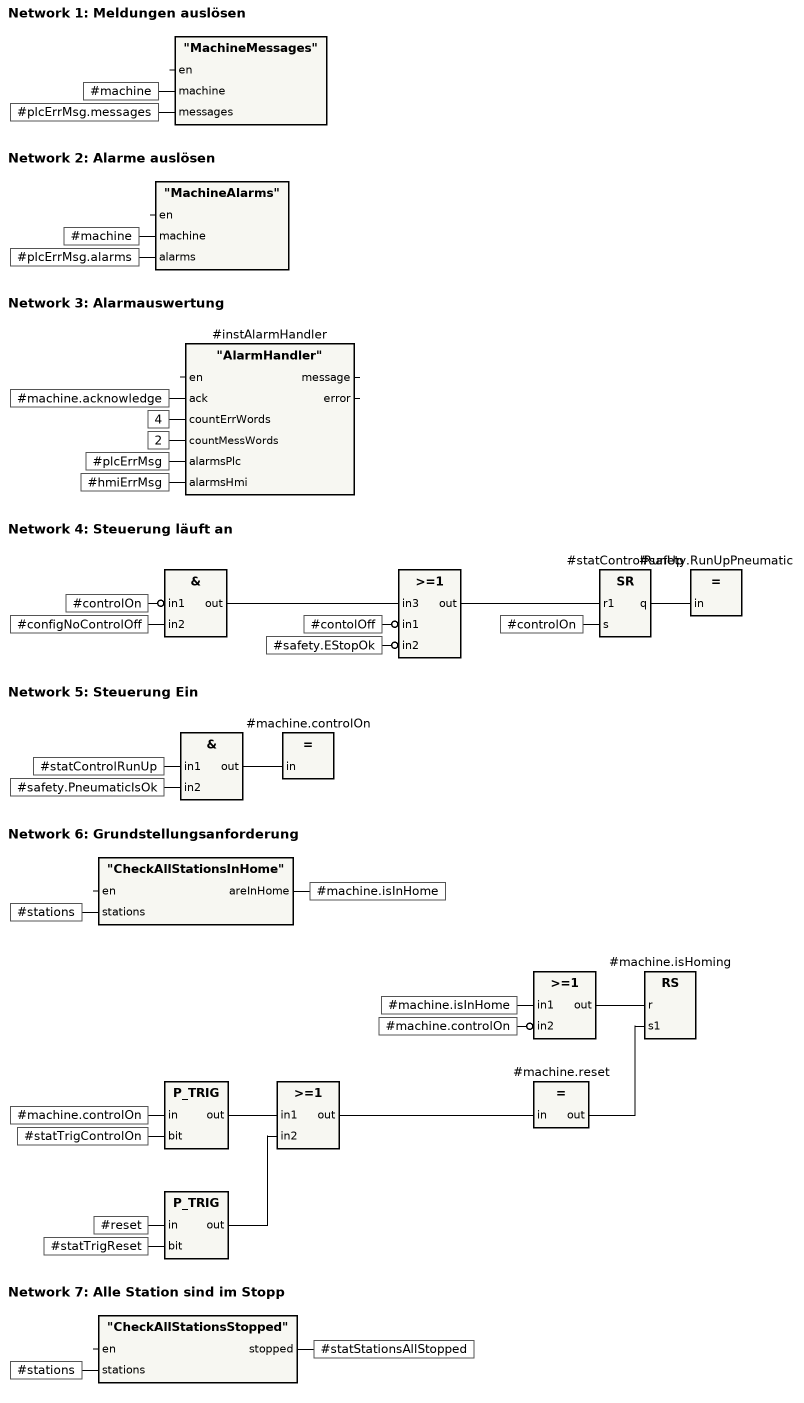
   "MachineMessages"(machine := #machine, messages := #plcErrMsg.messages);
END_REGION

REGION Network 2: Alarme auslösen
   "MachineAlarms"(machine := #machine, alarms := #plcErrMsg.alarms);
END_REGION

REGION Network 3: Alarmauswertung
   #instAlarmHandler(ack := #machine.acknowledge,   // "AlarmHandler"
                     countErrWords := 4,
                     countMessWords := 2,
                     alarmsPlc := #plcErrMsg,
                     alarmsHmi := #hmiErrMsg);
END_REGION

REGION Network 4: Steuerung läuft an
   IF #controlOn THEN
       #statControlRunUp := TRUE;   // SR flip-flop
   END_IF;
   IF (NOT #controlOn AND #configNoControlOff) OR NOT #contolOff OR NOT #safety.EStopOk THEN
       #statControlRunUp := FALSE;
   END_IF;
   #safety.RunUpPneumatic := #statControlRunUp;
END_REGION

REGION Network 5: Steuerung Ein
   #machine.controlOn := #statControlRunUp AND #safety.PneumaticIsOk;
END_REGION

REGION Network 6: Grundstellungsanforderung
   "CheckAllStationsInHome"(stations := #stations, areInHome => #machine.isInHome);
   #_w1 := #machine.controlOn AND NOT #statTrigControlOn;   // rising edge
   #statTrigControlOn := #machine.controlOn;
   #_w2 := #reset AND NOT #statTrigReset;   // rising edge
   #statTrigReset := #reset;
   #machine.reset := #_w1 OR #_w2;
   IF #machine.isInHome OR NOT #machine.controlOn THEN
       #machine.isHoming := FALSE;   // RS flip-flop
   END_IF;
   IF #machine.reset THEN #machine.isHoming := TRUE; END_IF;
END_REGION

REGION Network 7: Alle Station sind im Stopp
   "CheckAllStationsStopped"(stations := #stations, stopped => #statStationsAllStopped);
END_REGION

REGION Network 8: Automatikmodus
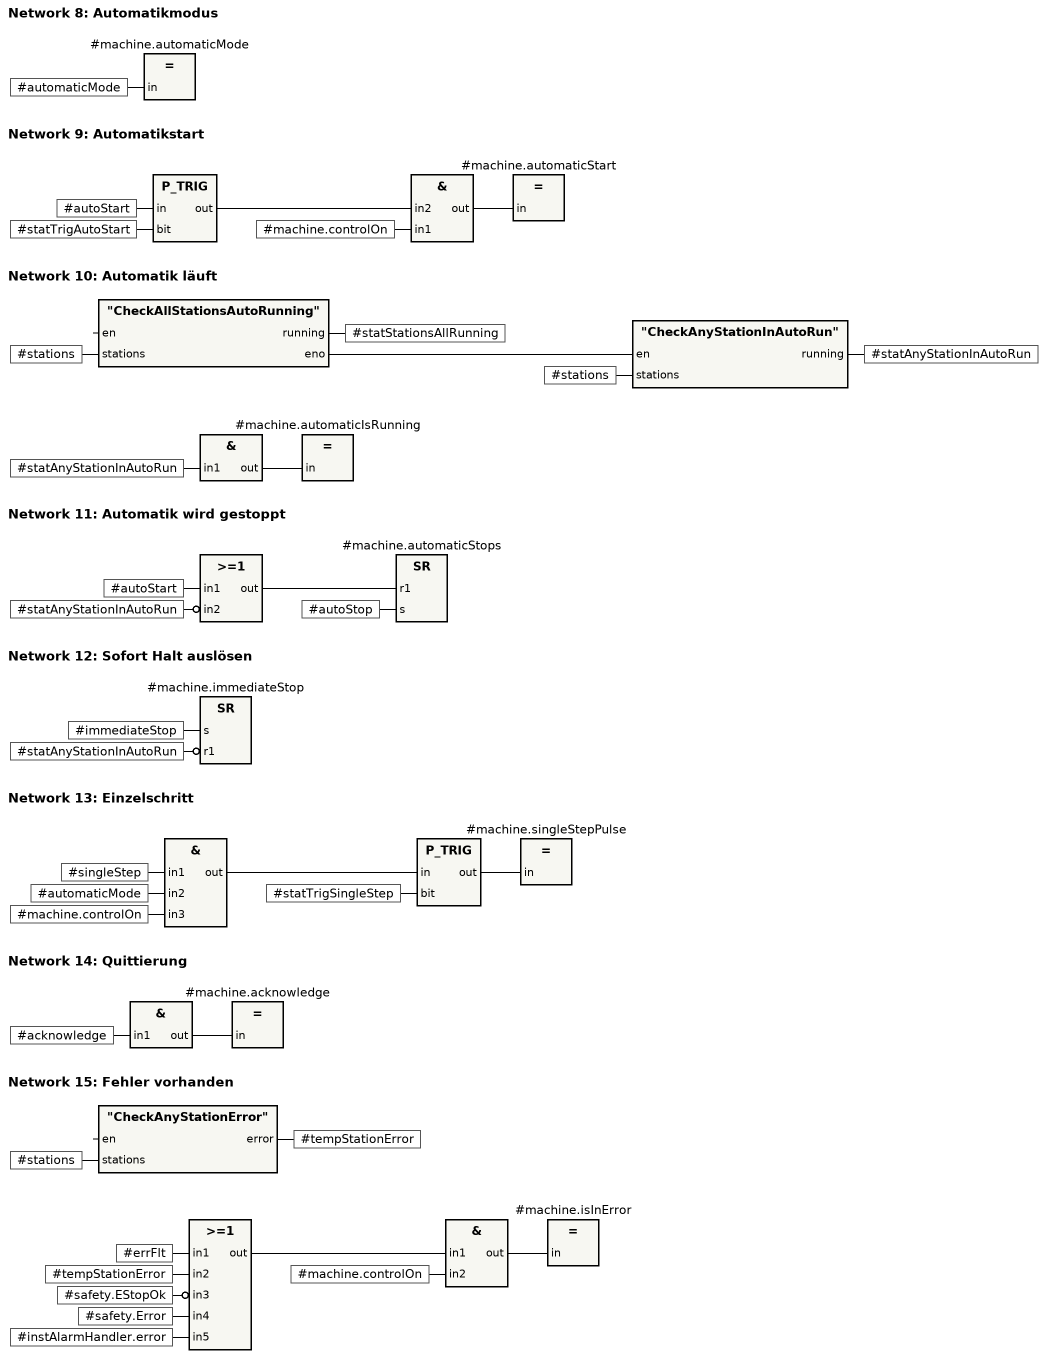
   #machine.automaticMode := #automaticMode;
END_REGION

REGION Network 9: Automatikstart
   #_w1 := #autoStart AND NOT #statTrigAutoStart;   // rising edge
   #statTrigAutoStart := #autoStart;
   #machine.automaticStart := #_w1 AND #machine.controlOn;
END_REGION

REGION Network 10: Automatik läuft
   "CheckAllStationsAutoRunning"(stations := #stations, running => #statStationsAllRunning, ENO => #_w1);
   IF #_w1 THEN
       "CheckAnyStationInAutoRun"(stations := #stations, running => #statAnyStationInAutoRun);
   END_IF;
   #machine.automaticIsRunning := #statAnyStationInAutoRun;
END_REGION

REGION Network 11: Automatik wird gestoppt
   IF #autoStop THEN
       #machine.automaticStops := TRUE;   // SR flip-flop
   END_IF;
   IF #autoStart OR NOT #statAnyStationInAutoRun THEN #machine.automaticStops := FALSE; END_IF;
END_REGION

REGION Network 12: Sofort Halt auslösen
   IF #immediateStop THEN
       #machine.immediateStop := TRUE;   // SR flip-flop
   END_IF;
   IF NOT #statAnyStationInAutoRun THEN #machine.immediateStop := FALSE; END_IF;
END_REGION

REGION Network 13: Einzelschritt
   #_w1 := #singleStep AND #automaticMode AND #machine.controlOn;
   #_w2 := #_w1 AND NOT #statTrigSingleStep;   // rising edge
   #statTrigSingleStep := #_w1;
   #machine.singleStepPulse := #_w2;
END_REGION

REGION Network 14: Quittierung
   #machine.acknowledge := #acknowledge;
END_REGION

REGION Network 15: Fehler vorhanden
   "CheckAnyStationError"(stations := #stations, error => #tempStationError);
   #machine.isInError := (#errFlt OR #tempStationError OR NOT #safety.EStopOk OR #safety.Error OR #instAlarmHandler.error) AND #machine.controlOn;
END_REGION

REGION Network 16: Initialisierung Bewegungsfunktionen (Teil 1)
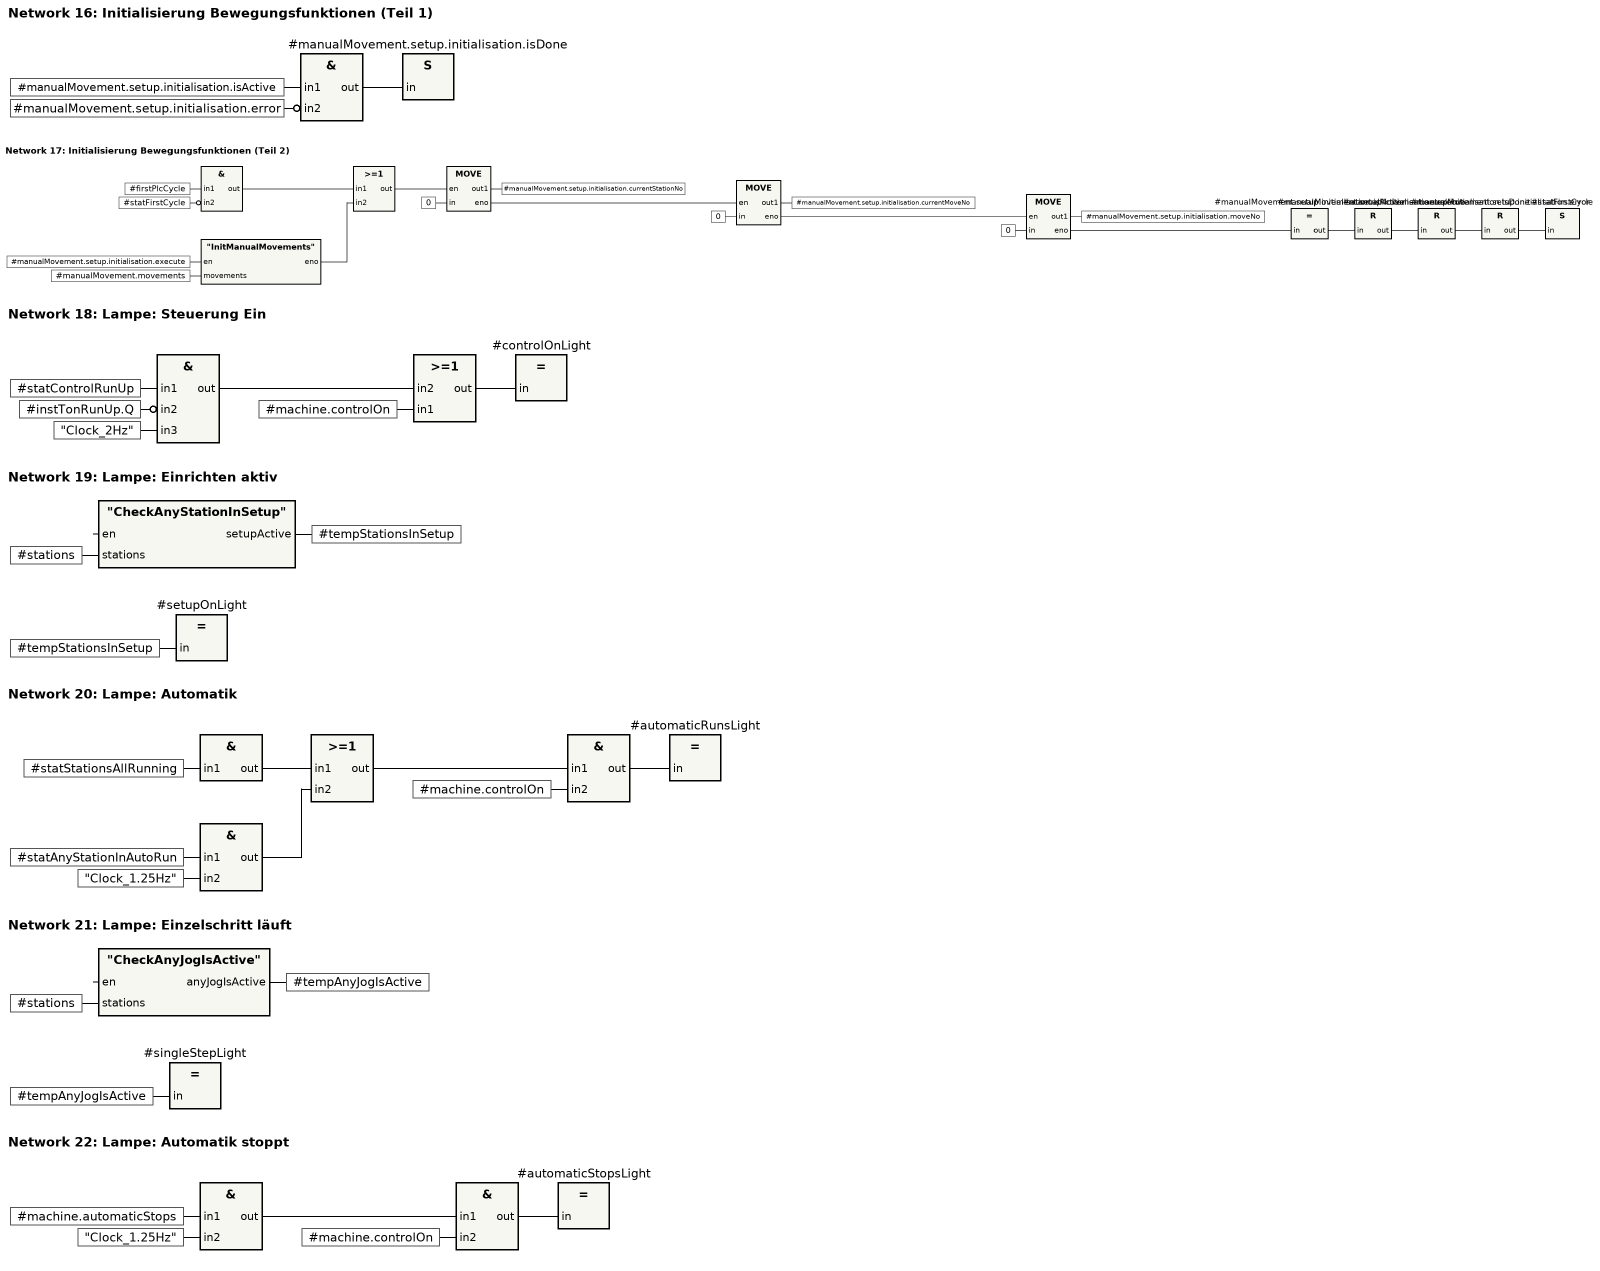
   IF #manualMovement.setup.initialisation.isActive AND NOT #manualMovement.setup.initialisation.error THEN
       #manualMovement.setup.initialisation.isDone := TRUE;
   END_IF;
END_REGION

REGION Network 17: Initialisierung Bewegungsfunktionen (Teil 2)
   "InitManualMovements"(EN := #manualMovement.setup.initialisation.execute,
                         movements := #manualMovement.movements,
                         ENO => #_w1);
   #_w2 := (#firstPlcCycle AND NOT #statFirstCycle) OR #_w1;
   IF #_w2 THEN
       #manualMovement.setup.initialisation.currentStationNo := 0;
       #manualMovement.setup.initialisation.currentMoveNo := 0;
       #manualMovement.setup.initialisation.moveNo := 0;
   END_IF;
   #manualMovement.setup.initialisation.isActive := #_w2;
   IF #_w2 THEN
       #manualMovement.setup.initialisation.execute := FALSE;
       #manualMovement.setup.initialisation.isDone := FALSE;
       #manualMovement.setup.initialisation.error := FALSE;
       #statFirstCycle := TRUE;
   END_IF;
END_REGION

REGION Network 18: Lampe: Steuerung Ein
   #controlOnLight := (#statControlRunUp AND NOT #instTonRunUp.Q AND "Clock_2Hz") OR #machine.controlOn;
END_REGION

REGION Network 19: Lampe: Einrichten aktiv
   "CheckAnyStationInSetup"(stations := #stations, setupActive => #tempStationsInSetup);
   #setupOnLight := #tempStationsInSetup;
END_REGION

REGION Network 20: Lampe: Automatik
   #automaticRunsLight := (#statStationsAllRunning OR (#statAnyStationInAutoRun AND "Clock_1.25Hz")) AND #machine.controlOn;
END_REGION

REGION Network 21: Lampe: Einzelschritt läuft
   "CheckAnyJogIsActive"(stations := #stations, anyJogIsActive => #tempAnyJogIsActive);
   #singleStepLight := #tempAnyJogIsActive;
END_REGION

REGION Network 22: Lampe: Automatik stoppt
   #automaticStopsLight := #machine.automaticStops AND "Clock_1.25Hz" AND #machine.controlOn;
END_REGION

REGION Network 23: Lampe: Fehler
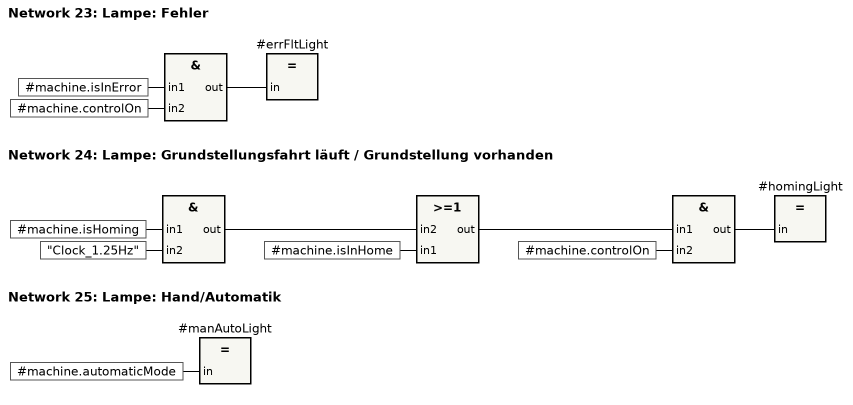
   #errFltLight := #machine.isInError AND #machine.controlOn;
END_REGION

REGION Network 24: Lampe: Grundstellungsfahrt läuft / Grundstellung vorhanden
   #homingLight := ((#machine.isHoming AND "Clock_1.25Hz") OR #machine.isInHome) AND #machine.controlOn;
END_REGION

REGION Network 25: Lampe: Hand/Automatik
   #manAutoLight := #machine.automaticMode;
END_REGION
END_FUNCTION_BLOCK

FUNCTION_BLOCK "StationControl"   // FB9001, FBD
TITLE = Steuerung Station
{ S7_Optimized_Access := 'TRUE' }
VERSION : 0.1
// Ersteller: Andreas Fast Automation
// E-Mail: automation@fast-andreas.de
// 
// Projekt dient zu Demonstrationszwecken und frei genutzt werden.
// 
// Bausteinbeschreibung:
   VAR_INPUT
      stationNo : Int := 1;   // Stationsnummer
      safetyOk : Bool;   // Schutzkreis geschlossen
      autoStart : Bool;   // Automatikstart
      autoStop : Bool;   // Automatikstopp
      singlePulse : Bool;   // Einzelschritt (Halbautomatik)
      reset : Bool;   // Station rücksetzen/Grundstellungsfahrt starten
      ack : Bool;   // Quittieren
      error : Bool;   // Störung vorhanden
      robotsStopped : Bool := true;   // Roboter sind angehalten
   END_VAR
   VAR_IN_OUT
      exists : Bool;   // Station existiert
      machine : "typeMachine";
      station : "typeStationSignals";
      stepSeqs : "typeStepSequences";
      setup : "typeManualMoveSetup";
      plcErrMsg : "typePlcErrMsg";
      hmiErrMsg : "typeHmiErrMsg";
   END_VAR
   VAR
      statTrigReset : Bool;
      statTrigSinglePulse : Bool;
      statTrigHomingDone : Bool;
      sxTrigAutomaticMode : Bool;
      sxTrigTap : Bool;
      sxTrigAuto : Bool;
      instAlarmHandler : "AlarmHandler";
      tonTEST : TON_TIME;
   END_VAR
   VAR_TEMP
      tempHomingDone : Bool;
      tempSqInError : Bool;
      tempSqAllInHome : Bool;
      tempSqAllJogDone : Bool;
      tempSqsAreWaitingOrInError : Bool;
      tempResetReleaseCycle : Bool;
      tempSinglePulse : Bool;
   END_VAR
   VAR_TEMP   // added for the SCL form of the ladder/FBD networks
      _w1 : Bool;
      _w2 : Bool;
      _w3 : Bool;
   END_VAR
BEGIN

REGION Network 1: Station ist vorhanden / nicht reserviert
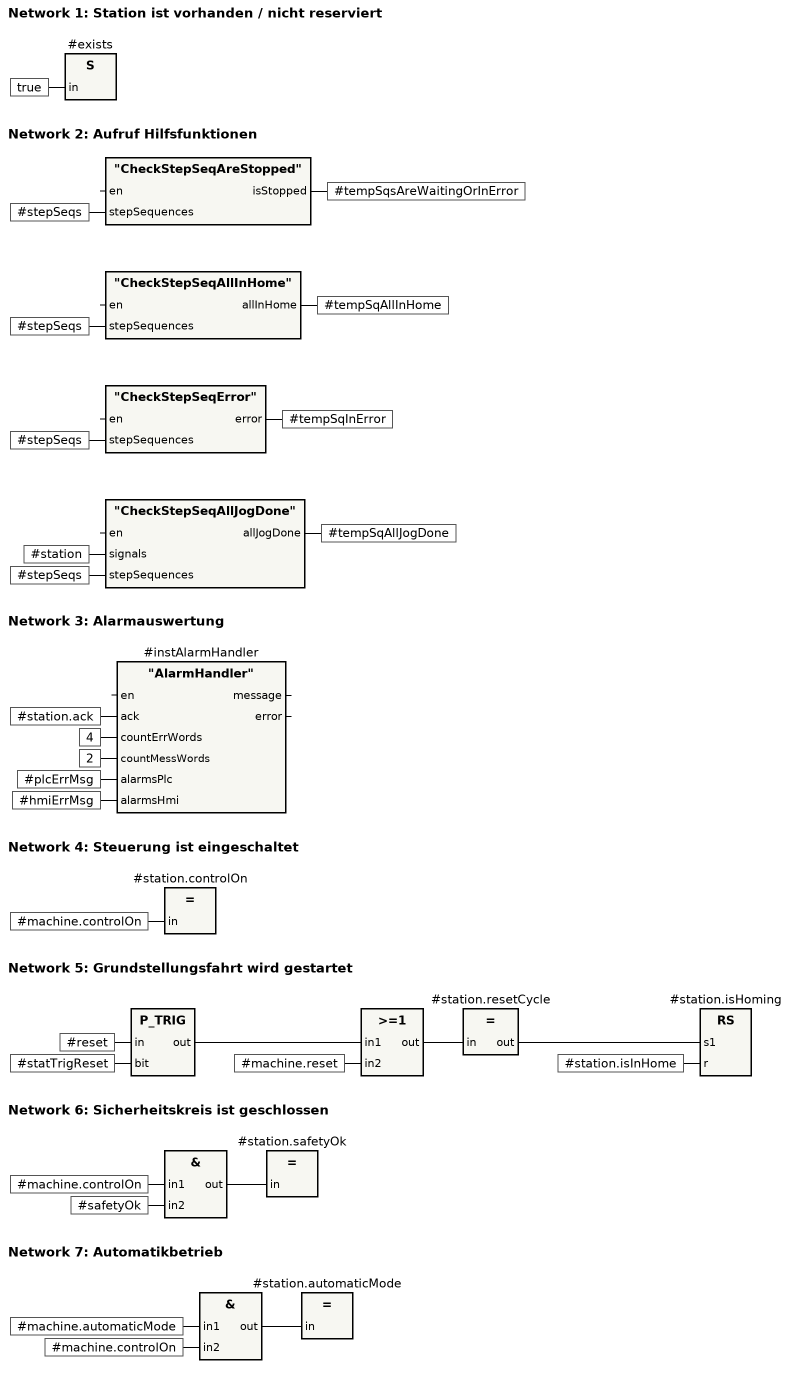
   IF true THEN #exists := TRUE; END_IF;
END_REGION

REGION Network 2: Aufruf Hilfsfunktionen
   "CheckStepSeqAreStopped"(stepSequences := #stepSeqs, isStopped => #tempSqsAreWaitingOrInError);
   "CheckStepSeqAllInHome"(stepSequences := #stepSeqs, allInHome => #tempSqAllInHome);
   "CheckStepSeqError"(stepSequences := #stepSeqs, error => #tempSqInError);
   "CheckStepSeqAllJogDone"(signals := #station, stepSequences := #stepSeqs, allJogDone => #tempSqAllJogDone);
END_REGION

REGION Network 3: Alarmauswertung
   #instAlarmHandler(ack := #station.ack,   // "AlarmHandler"
                     countErrWords := 4,
                     countMessWords := 2,
                     alarmsPlc := #plcErrMsg,
                     alarmsHmi := #hmiErrMsg);
END_REGION

REGION Network 4: Steuerung ist eingeschaltet
   #station.controlOn := #machine.controlOn;
END_REGION

REGION Network 5: Grundstellungsfahrt wird gestartet
   #_w1 := #reset AND NOT #statTrigReset;   // rising edge
   #statTrigReset := #reset;
   #station.resetCycle := #_w1 OR #machine.reset;
   IF #station.isInHome THEN
       #station.isHoming := FALSE;   // RS flip-flop
   END_IF;
   IF #station.resetCycle THEN #station.isHoming := TRUE; END_IF;
END_REGION

REGION Network 6: Sicherheitskreis ist geschlossen
   #station.safetyOk := #machine.controlOn AND #safetyOk;
END_REGION

REGION Network 7: Automatikbetrieb
   #station.automaticMode := #machine.automaticMode AND #machine.controlOn;
END_REGION

REGION Network 8: Handbetrieb
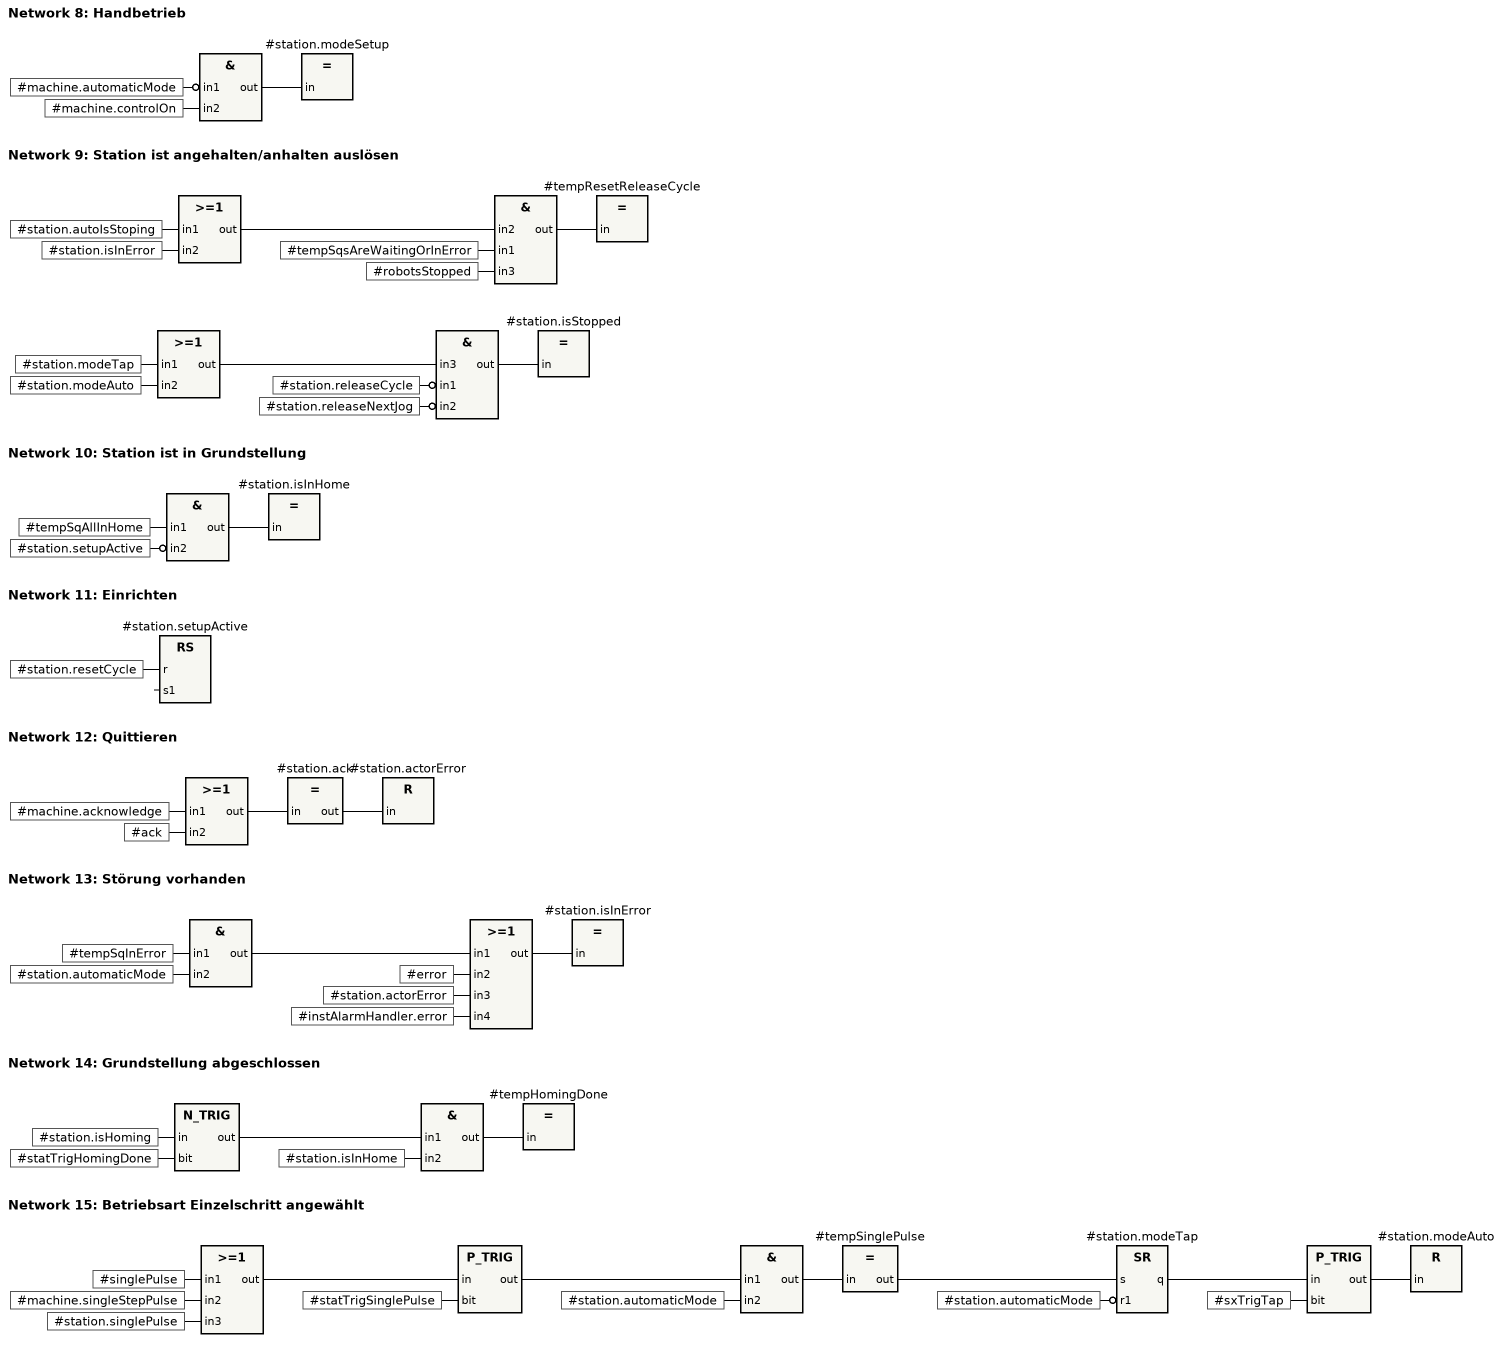
   #station.modeSetup := NOT #machine.automaticMode AND #machine.controlOn;
END_REGION

REGION Network 9: Station ist angehalten/anhalten auslösen
   #tempResetReleaseCycle := (#station.autoIsStoping OR #station.isInError) AND #tempSqsAreWaitingOrInError AND #robotsStopped;
   #station.isStopped := (#station.modeTap OR #station.modeAuto) AND NOT #station.releaseCycle AND NOT #station.releaseNextJog;
END_REGION

REGION Network 10: Station ist in Grundstellung
   #station.isInHome := #tempSqAllInHome AND NOT #station.setupActive;
END_REGION

REGION Network 11: Einrichten
   IF #station.resetCycle THEN
       #station.setupActive := FALSE;   // RS flip-flop
   END_IF;
END_REGION

REGION Network 12: Quittieren
   #station.ack := #machine.acknowledge OR #ack;
   IF #station.ack THEN #station.actorError := FALSE; END_IF;
END_REGION

REGION Network 13: Störung vorhanden
   #station.isInError := (#tempSqInError AND #station.automaticMode) OR #error OR #station.actorError OR #instAlarmHandler.error;
END_REGION

REGION Network 14: Grundstellung abgeschlossen
   #_w1 := NOT #station.isHoming AND #statTrigHomingDone;   // falling edge
   #statTrigHomingDone := #station.isHoming;
   #tempHomingDone := #_w1 AND #station.isInHome;
END_REGION

REGION Network 15: Betriebsart Einzelschritt angewählt
   #_w1 := #singlePulse OR #machine.singleStepPulse OR #station.singlePulse;
   #_w2 := #_w1 AND NOT #statTrigSinglePulse;   // rising edge
   #statTrigSinglePulse := #_w1;
   #tempSinglePulse := #_w2 AND #station.automaticMode;
   IF #tempSinglePulse THEN
       #station.modeTap := TRUE;   // SR flip-flop
   END_IF;
   IF NOT #station.automaticMode THEN #station.modeTap := FALSE; END_IF;
   #_w3 := #station.modeTap AND NOT #sxTrigTap;   // rising edge
   #sxTrigTap := #station.modeTap;
   IF #_w3 THEN #station.modeAuto := FALSE; END_IF;
END_REGION

REGION Network 16: Betriebsart Automatikbetrieb angewählt
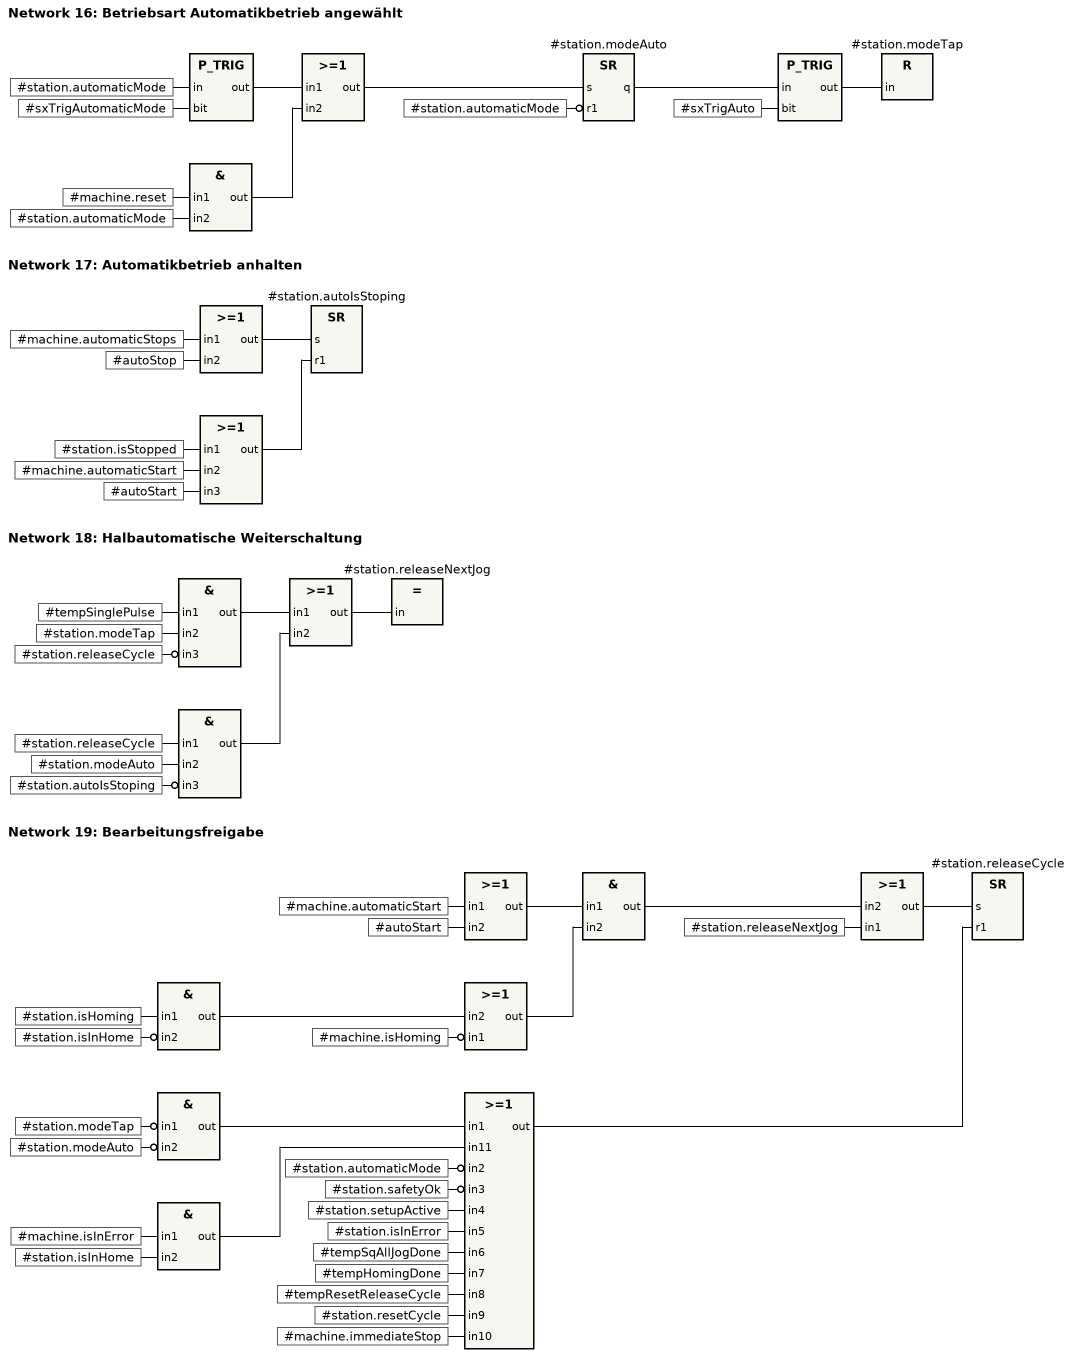
   #_w1 := #station.automaticMode AND NOT #sxTrigAutomaticMode;   // rising edge
   #sxTrigAutomaticMode := #station.automaticMode;
   IF #_w1 OR (#machine.reset AND #station.automaticMode) THEN
       #station.modeAuto := TRUE;   // SR flip-flop
   END_IF;
   IF NOT #station.automaticMode THEN #station.modeAuto := FALSE; END_IF;
   #_w2 := #station.modeAuto AND NOT #sxTrigAuto;   // rising edge
   #sxTrigAuto := #station.modeAuto;
   IF #_w2 THEN #station.modeTap := FALSE; END_IF;
END_REGION

REGION Network 17: Automatikbetrieb anhalten
   IF #machine.automaticStops OR #autoStop THEN
       #station.autoIsStoping := TRUE;   // SR flip-flop
   END_IF;
   IF #station.isStopped OR #machine.automaticStart OR #autoStart THEN
       #station.autoIsStoping := FALSE;
   END_IF;
END_REGION

REGION Network 18: Halbautomatische Weiterschaltung
   #station.releaseNextJog := (#tempSinglePulse AND #station.modeTap AND NOT #station.releaseCycle) OR (#station.releaseCycle AND #station.modeAuto AND NOT #station.autoIsStoping);
END_REGION

REGION Network 19: Bearbeitungsfreigabe
   IF ((#machine.automaticStart OR #autoStart) AND ((#station.isHoming AND NOT #station.isInHome) OR NOT #machine.isHoming)) OR #station.releaseNextJog THEN
       #station.releaseCycle := TRUE;   // SR flip-flop
   END_IF;
   IF (NOT #station.modeTap AND NOT #station.modeAuto) OR (#machine.isInError AND #station.isInHome) OR NOT #station.automaticMode OR NOT #station.safetyOk OR #station.setupActive OR #station.isInError OR #tempSqAllJogDone OR #tempHomingDone OR #tempResetReleaseCycle OR #station.resetCycle OR #machine.immediateStop THEN
       #station.releaseCycle := FALSE;
   END_IF;
END_REGION

REGION Network 20: Initialisierung für Einrichtbewegungen
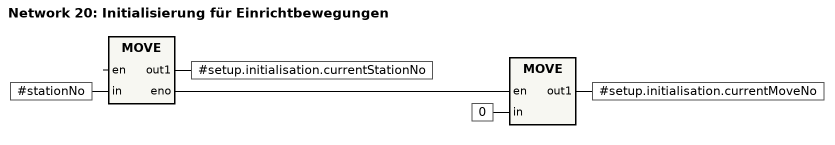
   #setup.initialisation.currentStationNo := #stationNo;
   #setup.initialisation.currentMoveNo := 0;
END_REGION
END_FUNCTION_BLOCK

FUNCTION_BLOCK "AlarmHandler"   // FB9009, SCL
{ S7_Optimized_Access := 'TRUE' }
VERSION : 0.1
   VAR_INPUT
      ack : Bool;   // Quittierung
      countErrWords : Int := 4;   // Anzahl Fehlermelde-Wörter
      countMessWords : Int;
   END_VAR
   VAR_OUTPUT
      message : Bool;
      error : Bool;   // Mindestens ein Fehler steht an
   END_VAR
   VAR_IN_OUT
      alarmsPlc : "typePlcErrMsg";
      alarmsHmi : "typeHmiErrMsg";
   END_VAR
   VAR
      risAck : Bool;
      instRisTrigger : R_TRIG;
      instTpAck : TP_TIME;
   END_VAR
   VAR_TEMP
      ackPulse : Bool;
      i : Int;
      x : Int;
      lengthPlcErrors : Int;
      lengthPlcMessages : Int;
   END_VAR
BEGIN
   // Ersteller: Andreas Fast Automation
   // E-Mail: automation@fast-andreas.de
   //
   // Projekt dient zu Demonstrationszwecken und frei genutzt werden.
   //
   // Bausteinbeschreibung:
   // 

   // Init values
   #lengthPlcErrors := #countErrWords * 16;
   #lengthPlcMessages := #countMessWords * 16;

   #instRisTrigger(CLK := #ack,
                   Q => #risAck);


   #instTpAck(IN:=#risAck,
              PT:=t#1s,
              Q=>#ackPulse);

   // Acknowledge signals for HMI
   FOR #i := 1 TO #countErrWords DO
       IF #ackPulse THEN
           #alarmsHmi.alarmAckPlc[#i + #countErrWords] := 16#FFFF;
       ELSE
           #alarmsHmi.alarmAckPlc[#i + #countErrWords] := 16#0;
       END_IF;
   END_FOR;


   // Clear errors of PLC
   IF #risAck THEN
       FOR #i := 1 TO #lengthPlcErrors DO
           #alarmsPlc.alarms.errorNo[#i] := FALSE;
       END_FOR;
   END_IF;

   // Assign plc alarms to HMI triggers
   FOR #i := 1 TO #countErrWords DO
       #x := (#i - 1) * 16;

       #alarmsHmi.alarmAckPlc[#i].%X0 := #alarmsPlc.alarms.errorNo[#x + 1];
       #alarmsHmi.alarmAckPlc[#i].%X1 := #alarmsPlc.alarms.errorNo[#x + 2];
       #alarmsHmi.alarmAckPlc[#i].%X2 := #alarmsPlc.alarms.errorNo[#x + 3];
       #alarmsHmi.alarmAckPlc[#i].%X3 := #alarmsPlc.alarms.errorNo[#x + 4];
       #alarmsHmi.alarmAckPlc[#i].%X4 := #alarmsPlc.alarms.errorNo[#x + 5];
       #alarmsHmi.alarmAckPlc[#i].%X5 := #alarmsPlc.alarms.errorNo[#x + 6];
       #alarmsHmi.alarmAckPlc[#i].%X6 := #alarmsPlc.alarms.errorNo[#x + 7];
       #alarmsHmi.alarmAckPlc[#i].%X7 := #alarmsPlc.alarms.errorNo[#x + 8];
       #alarmsHmi.alarmAckPlc[#i].%X8 := #alarmsPlc.alarms.errorNo[#x + 9];
       #alarmsHmi.alarmAckPlc[#i].%X9 := #alarmsPlc.alarms.errorNo[#x + 10];
       #alarmsHmi.alarmAckPlc[#i].%X10 := #alarmsPlc.alarms.errorNo[#x + 11];
       #alarmsHmi.alarmAckPlc[#i].%X11 := #alarmsPlc.alarms.errorNo[#x + 12];
       #alarmsHmi.alarmAckPlc[#i].%X12 := #alarmsPlc.alarms.errorNo[#x + 13];
       #alarmsHmi.alarmAckPlc[#i].%X13 := #alarmsPlc.alarms.errorNo[#x + 14];
       #alarmsHmi.alarmAckPlc[#i].%X14 := #alarmsPlc.alarms.errorNo[#x + 15];
       #alarmsHmi.alarmAckPlc[#i].%X15 := #alarmsPlc.alarms.errorNo[#x + 16];
   END_FOR;

   // Assign PLC messages to HMI messages
   FOR #i := 1 TO #countMessWords DO
       #x := (#i - 1) * 16;

       #alarmsHmi.message[#i].%X0 := #alarmsPlc.messages.msgNo[#x + 1];
       #alarmsHmi.message[#i].%X1 := #alarmsPlc.messages.msgNo[#x + 2];
       #alarmsHmi.message[#i].%X2 := #alarmsPlc.messages.msgNo[#x + 3];
       #alarmsHmi.message[#i].%X3 := #alarmsPlc.messages.msgNo[#x + 4];
       #alarmsHmi.message[#i].%X4 := #alarmsPlc.messages.msgNo[#x + 5];
       #alarmsHmi.message[#i].%X5 := #alarmsPlc.messages.msgNo[#x + 6];
       #alarmsHmi.message[#i].%X6 := #alarmsPlc.messages.msgNo[#x + 7];
       #alarmsHmi.message[#i].%X7 := #alarmsPlc.messages.msgNo[#x + 8];
       #alarmsHmi.message[#i].%X8 := #alarmsPlc.messages.msgNo[#x + 9];
       #alarmsHmi.message[#i].%X9 := #alarmsPlc.messages.msgNo[#x + 10];
       #alarmsHmi.message[#i].%X10 := #alarmsPlc.messages.msgNo[#x + 11];
       #alarmsHmi.message[#i].%X11 := #alarmsPlc.messages.msgNo[#x + 12];
       #alarmsHmi.message[#i].%X12 := #alarmsPlc.messages.msgNo[#x + 13];
       #alarmsHmi.message[#i].%X13 := #alarmsPlc.messages.msgNo[#x + 14];
       #alarmsHmi.message[#i].%X14 := #alarmsPlc.messages.msgNo[#x + 15];
       #alarmsHmi.message[#i].%X15 := #alarmsPlc.messages.msgNo[#x + 16];
   END_FOR;



   // set error 
   #error := false;
   FOR #i := 1 TO #lengthPlcErrors DO
       IF #alarmsPlc.alarms.errorNo[#i] THEN
           #error:= TRUE;
           EXIT;
       END_IF;
   END_FOR;


   // set message
   #message := false;
   FOR #i := 1 TO #lengthPlcMessages DO
       IF #alarmsPlc.messages.msgNo[#i] THEN
           #message := TRUE;
           EXIT;
       END_IF;
   END_FOR;
END_FUNCTION_BLOCK

// folder: 9. Library/9.1 Framework Functions

FUNCTION "SetError" : Void   // FC900, FBD
TITLE = Setze Fehler
{ S7_Optimized_Access := 'TRUE' }
VERSION : 0.1
// Ersteller: Andreas Fast Automation
// E-Mail: automation@fast-andreas.de
// 
// Projekt dient zu Demonstrationszwecken und frei genutzt werden.
// 
// Bausteinbeschreibung:
   VAR_INPUT
      trigger : Bool;   // Auslöser
      logic : Bool;   // Auslöserlogik; 0 = trigger ausgelöst bei false
   END_VAR
   VAR_OUTPUT
      error : Bool;
   END_VAR
BEGIN

REGION Network 1
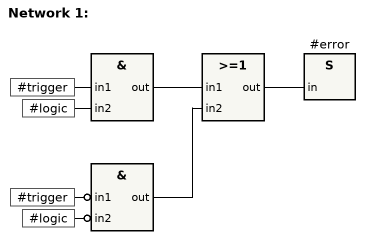
   IF (#trigger AND #logic) OR (NOT #trigger AND NOT #logic) THEN #error := TRUE; END_IF;
END_REGION
END_FUNCTION

FUNCTION "CheckAllStationsStopped" : Void   // FC901, SCL
{ S7_Optimized_Access := 'TRUE' }
VERSION : 0.1
   VAR_OUTPUT
      stopped : Bool;   // All stations are stopped
   END_VAR
   VAR_IN_OUT
      stations : "typeStations";
   END_VAR
   VAR_TEMP
      tempCounter : USInt;
   END_VAR
BEGIN
   // Ersteller: Andreas Fast Automation
   // E-Mail: automation@fast-andreas.de
   //
   // Projekt dient zu Demonstrationszwecken und frei genutzt werden.
   //
   // Bausteinbeschreibung:
   // 

   #stopped := true;

   FOR #tempCounter := 1 TO "SYS_MACHINE_MAXSTATIONS" DO
       // Check if all stations are stopped
       IF NOT #stations.station[#tempCounter].signals.isStopped AND #stations.station[#tempCounter].exists THEN
           #stopped := false;
           RETURN;
       END_IF;
   END_FOR;
END_FUNCTION

FUNCTION "CheckAnyStationError" : Void   // FC902, SCL
{ S7_Optimized_Access := 'TRUE' }
VERSION : 0.1
// Check if any station is in error
   VAR_OUTPUT
      error : Bool;
   END_VAR
   VAR_IN_OUT
      stations : "typeStations";
   END_VAR
   VAR_TEMP
      tempCounter : USInt;
   END_VAR
BEGIN
   // Ersteller: Andreas Fast Automation
   // E-Mail: automation@fast-andreas.de
   //
   // Projekt dient zu Demonstrationszwecken und frei genutzt werden.
   //
   // Bausteinbeschreibung:
   // 

   #error := false;

   FOR #tempCounter := 1 TO "SYS_MACHINE_MAXSTATIONS" DO
       // Check for error in stations
       IF #stations.station[#tempCounter].signals.isInError AND #stations.station[#tempCounter].exists THEN
           #error := true;
           RETURN;
       END_IF;
   END_FOR;
END_FUNCTION

FUNCTION "CheckAnyStationInSetup" : Void   // FC903, SCL
{ S7_Optimized_Access := 'TRUE' }
VERSION : 0.1
// Check if any station is in error
   VAR_OUTPUT
      setupActive : Bool;
   END_VAR
   VAR_IN_OUT
      stations : "typeStations";
   END_VAR
   VAR_TEMP
      tempCounter : USInt;
   END_VAR
BEGIN
   // Ersteller: Andreas Fast Automation
   // E-Mail: automation@fast-andreas.de
   //
   // Projekt dient zu Demonstrationszwecken und frei genutzt werden.
   //
   // Bausteinbeschreibung:
   // 

   #setupActive := false;

   FOR #tempCounter := 1 TO "SYS_MACHINE_MAXSTATIONS" DO
       // Check for error in stations
       IF #stations.station[#tempCounter].signals.setupActive AND #stations.station[#tempCounter].exists THEN
           #setupActive := true;
           RETURN;
       END_IF;
   END_FOR;
END_FUNCTION

FUNCTION "CheckAllStationsInHome" : Void   // FC904, SCL
{ S7_Optimized_Access := 'TRUE' }
VERSION : 0.1
   VAR_OUTPUT
      areInHome : Bool;   // All stations are in home
   END_VAR
   VAR_IN_OUT
      stations : "typeStations";
   END_VAR
   VAR_TEMP
      tempCounter : USInt;
   END_VAR
BEGIN
   // Ersteller: Andreas Fast Automation
   // E-Mail: automation@fast-andreas.de
   //
   // Projekt dient zu Demonstrationszwecken und frei genutzt werden.
   //
   // Bausteinbeschreibung:
   // 

   #areInHome := true;

   FOR #tempCounter := 1 TO "SYS_MACHINE_MAXSTATIONS" DO
       // Check if all stations are stopped
       IF NOT #stations.station[#tempCounter].signals.isInHome AND #stations.station[#tempCounter].exists THEN
           #areInHome := false;
           RETURN ;
       END_IF;
   END_FOR;
END_FUNCTION

FUNCTION "CheckAllStationsAutoRunning" : Void   // FC905, SCL
{ S7_Optimized_Access := 'TRUE' }
VERSION : 0.1
   VAR_OUTPUT
      running : Bool;   // All stations in automatic run
   END_VAR
   VAR_IN_OUT
      stations : "typeStations";
   END_VAR
   VAR_TEMP
      tempCounter : USInt;
   END_VAR
BEGIN
   // Ersteller: Andreas Fast Automation
   // E-Mail: automation@fast-andreas.de
   //
   // Projekt dient zu Demonstrationszwecken und frei genutzt werden.
   //
   // Bausteinbeschreibung:
   // 

   #running := true;

   FOR #tempCounter := 1 TO "SYS_MACHINE_MAXSTATIONS" DO
       // Check if all stations are stopped
       IF NOT #stations.station[#tempCounter].signals.releaseCycle
           AND #stations.station[#tempCounter].exists
       THEN
           #running := false;
           RETURN;
       END_IF;
   END_FOR;
END_FUNCTION

FUNCTION "CheckAnyStationInAutoRun" : Void   // FC906, SCL
{ S7_Optimized_Access := 'TRUE' }
VERSION : 0.1
   VAR_OUTPUT
      running : Bool;   // All stations in automatic run
   END_VAR
   VAR_IN_OUT
      stations : "typeStations";
   END_VAR
   VAR_TEMP
      tempCounter : USInt;
   END_VAR
BEGIN
   // Ersteller: Andreas Fast Automation
   // E-Mail: automation@fast-andreas.de
   //
   // Projekt dient zu Demonstrationszwecken und frei genutzt werden.
   //
   // Bausteinbeschreibung:
   // 

   #running := false;

   FOR #tempCounter := 1 TO "SYS_MACHINE_MAXSTATIONS" DO
       // Check if all stations are stopped
       IF //#stations.station[#tempCounter].signals.modeAuto AND
           #stations.station[#tempCounter].signals.releaseCycle
           AND #stations.station[#tempCounter].exists
       THEN
           #running := true;
           RETURN;
       END_IF;
   END_FOR;
END_FUNCTION

FUNCTION "S7GraphParameters" : Void   // FC910, FBD
TITLE = Steuerung Graph Parameter
{ S7_Optimized_Access := 'TRUE' }
VERSION : 0.1
// Ersteller: Andreas Fast Automation
// E-Mail: automation@fast-andreas.de
// 
// Projekt dient zu Demonstrationszwecken und frei genutzt werden.
// 
// Bausteinbeschreibung:
   VAR_OUTPUT
      ack : Bool;   // Schrittkette quittieren
      init : Bool;   // Schrittkette in Initialschritt schalten
      auto : Bool;   // Automatikbetrieb
      man : Bool;   // Handbetrieb
      tap : Bool;   // Halbautomatischer Betrieb
      push : Bool;   // Schaltfreigabe für Transition im halbautomatischen Betrieb
   END_VAR
   VAR_IN_OUT
      signals : "typeStationSignals";
   END_VAR
BEGIN

REGION Network 1: Schrittkette in Initialschritt schalten
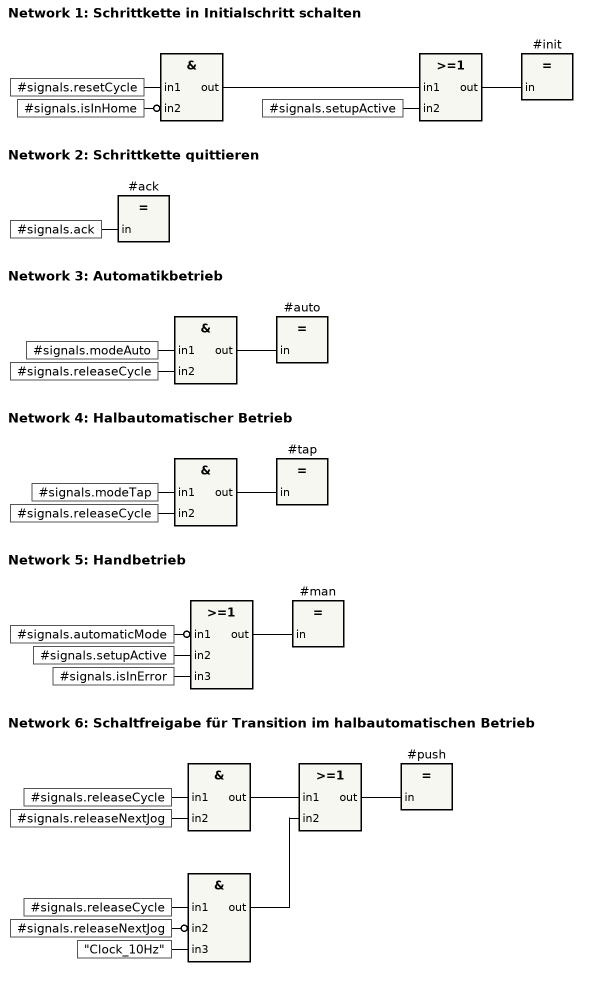
   #init := (#signals.resetCycle AND NOT #signals.isInHome) OR #signals.setupActive;
END_REGION

REGION Network 2: Schrittkette quittieren
   #ack := #signals.ack;
END_REGION

REGION Network 3: Automatikbetrieb
   #auto := #signals.modeAuto AND #signals.releaseCycle;
END_REGION

REGION Network 4: Halbautomatischer Betrieb
   #tap := #signals.modeTap AND #signals.releaseCycle;
END_REGION

REGION Network 5: Handbetrieb
   #man := NOT #signals.automaticMode OR #signals.setupActive OR #signals.isInError;
END_REGION

REGION Network 6: Schaltfreigabe für Transition im halbautomatischen Betrieb
   #push := (#signals.releaseCycle AND #signals.releaseNextJog) OR (#signals.releaseCycle AND NOT #signals.releaseNextJog AND "Clock_10Hz");
END_REGION
END_FUNCTION

FUNCTION "CheckStepSeqError" : Void   // FC911, SCL
{ S7_Optimized_Access := 'TRUE' }
VERSION : 0.1
   VAR_OUTPUT
      error : Bool;
   END_VAR
   VAR_IN_OUT
      stepSequences : "typeStepSequences";
   END_VAR
   VAR_TEMP
      tempCounter : USInt;
   END_VAR
BEGIN
   // Ersteller: Andreas Fast Automation
   // E-Mail: automation@fast-andreas.de
   //
   // Projekt dient zu Demonstrationszwecken und frei genutzt werden.
   //
   // Bausteinbeschreibung:
   // 

   #error := false;



   FOR #tempCounter := 1 TO "SYS_SQ_MAXSEQUENCES" DO
       // Check for error in stations
       IF #stepSequences.stepSeq[#tempCounter].error AND #stepSequences.stepSeq[#tempCounter].exists THEN
           #error := true;
           RETURN;
       END_IF;
   END_FOR;
END_FUNCTION

FUNCTION "CheckStepSeqAllInHome" : Void   // FC912, SCL
{ S7_Optimized_Access := 'TRUE' }
VERSION : 0.1
   VAR_OUTPUT
      allInHome : Bool;   // Alle Schrittketten in Grundstellung
   END_VAR
   VAR_IN_OUT
      stepSequences : "typeStepSequences";
   END_VAR
   VAR_TEMP
      tempCounter : USInt;
   END_VAR
BEGIN
   // Ersteller: Andreas Fast Automation
   // E-Mail: automation@fast-andreas.de
   //
   // Projekt dient zu Demonstrationszwecken und frei genutzt werden.
   //
   // Bausteinbeschreibung:
   // 

   #allInHome := true;



   FOR #tempCounter := 1 TO "SYS_SQ_MAXSEQUENCES" DO
       // Check for error in stations
       IF NOT #stepSequences.stepSeq[#tempCounter].inHome AND #stepSequences.stepSeq[#tempCounter].exists THEN
           #allInHome := false;
           RETURN;
       END_IF;
   END_FOR;
END_FUNCTION

FUNCTION "CheckStepSeqAreStopped" : Void   // FC913, SCL
{ S7_Optimized_Access := 'TRUE' }
VERSION : 0.1
   VAR_OUTPUT
      isStopped : Bool;
   END_VAR
   VAR_IN_OUT
      stepSequences : "typeStepSequences";
   END_VAR
   VAR_TEMP
      tempCounter : USInt;
   END_VAR
BEGIN
   // Ersteller: Andreas Fast Automation
   // E-Mail: automation@fast-andreas.de
   //
   // Projekt dient zu Demonstrationszwecken und frei genutzt werden.
   //
   // Bausteinbeschreibung:
   // 

   #isStopped := true;


   FOR #tempCounter := 1 TO "SYS_SQ_MAXSEQUENCES" DO
       // Check for error in stations
       IF NOT #stepSequences.stepSeq[#tempCounter].isWaiting AND NOT #stepSequences.stepSeq[#tempCounter].error AND #stepSequences.stepSeq[#tempCounter].exists THEN
           #isStopped := false;
           RETURN;
       END_IF;
   END_FOR;
END_FUNCTION

FUNCTION "CheckStepSeqAllJogDone" : Void   // FC914, SCL
{ S7_Optimized_Access := 'TRUE' }
VERSION : 0.1
   VAR_OUTPUT
      allJogDone : Bool;   // Alle Schrittketten haben halbautomatische Weiterschaltung abgeschlossen
   END_VAR
   VAR_IN_OUT
      signals : "typeStationSignals";
      stepSequences : "typeStepSequences";
   END_VAR
   VAR_TEMP
      tempCounter : USInt;
   END_VAR
BEGIN
   // Ersteller: Andreas Fast Automation
   // E-Mail: automation@fast-andreas.de
   //
   // Projekt dient zu Demonstrationszwecken und frei genutzt werden.
   //
   // Bausteinbeschreibung:
   // 

   #allJogDone := #signals.releaseCycle;

   IF #signals.modeTap AND NOT #signals.releaseNextJog OR (#signals.modeAuto AND #signals.autoIsStoping) THEN
       FOR #tempCounter := 1 TO "SYS_SQ_MAXSEQUENCES" DO
           // Check if step sequence is done and exists
           IF NOT #stepSequences.stepSeq[#tempCounter].jogDone AND NOT #stepSequences.stepSeq[#tempCounter].isWaiting  AND #stepSequences.stepSeq[#tempCounter].exists THEN
               #allJogDone := false;
               RETURN;
           END_IF;
       END_FOR;
   ELSE
       #allJogDone := false;
   END_IF;
END_FUNCTION

FUNCTION "CheckAnyJogIsActive" : Void   // FC915, SCL
{ S7_Optimized_Access := 'TRUE' }
VERSION : 0.1
   VAR_OUTPUT
      anyJogIsActive : Bool;   // Mindestens eine Schrittketten läuft noch in halbautomatischer Weiterschaltung
   END_VAR
   VAR_IN_OUT
      stations : "typeStations";
   END_VAR
   VAR_TEMP
      tempCounter : USInt;
   END_VAR
BEGIN
   // Ersteller: Andreas Fast Automation
   // E-Mail: automation@fast-andreas.de
   //
   // Projekt dient zu Demonstrationszwecken und frei genutzt werden.
   //
   // Bausteinbeschreibung:
   // 

   #anyJogIsActive := false;

   FOR #tempCounter := 1 TO "SYS_MACHINE_MAXSTATIONS" DO

       IF #stations.station[#tempCounter].exists AND
           #stations.station[#tempCounter].signals.modeTap AND
           #stations.station[#tempCounter].signals.releaseCycle
       THEN
           #anyJogIsActive := true;
           RETURN;
       END_IF;

   END_FOR;
END_FUNCTION

FUNCTION "S7GraphInterlock" : Void   // FC919, FBD
TITLE = S7G Verriegelung (notwendig für den Einzelschritt)
{ S7_Optimized_Access := 'TRUE' }
VERSION : 0.1
// Ersteller: Andreas Fast Automation
// E-Mail: automation@fast-andreas.de
// 
// Projekt dient zu Demonstrationszwecken und frei genutzt werden.
// 
// Bausteinbeschreibung:
   VAR_INPUT
      interlock : Bool;   // Verriegelung
      setting : Bool;   // Verriegelungslogik (interlock == setting -> out wird freigegeben)
      alarm : Bool;   // Beim Alarm wird out rückgesetzt
   END_VAR
   VAR_OUTPUT
      out : Bool;
   END_VAR
BEGIN

REGION Network 1
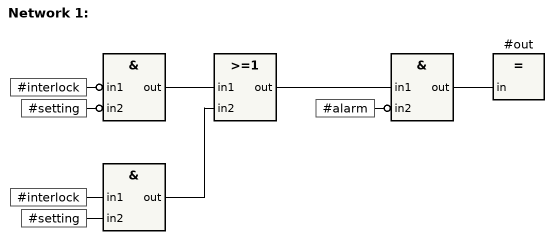
   #out := ((NOT #interlock AND NOT #setting) OR (#interlock AND #setting)) AND NOT #alarm;
END_REGION
END_FUNCTION

// folder: 9. Library/9.1 Framework Functions/ManualMovement

FUNCTION_BLOCK "ActorManualMovement"   // FB909, FBD
TITLE = Steuerung Einrichtbewegung eines Aktors
{ S7_Optimized_Access := 'TRUE' }
VERSION : 0.1
// Ersteller: Andreas Fast Automation
// E-Mail: automation@fast-andreas.de
// 
// Projekt dient zu Demonstrationszwecken und frei genutzt werden.
// 
// Bausteinbeschreibung:
   VAR_INPUT
      showValue : Bool;
      isExecutableRight : Bool;
      isExecutableLeft : Bool;
      showEndPositionRight : Bool;   // Sichtbarkeit rechte Seite
      showEndPositionLeft : Bool;   // Sichtbarkeit linke Seite
   END_VAR
   VAR_OUTPUT
      manualMoveNo : UInt;
   END_VAR
   VAR_IN_OUT
      manualWorkPos : Bool;   // Manueller Ansteuerbefehl für Arbeitsstellung
      manualHomePos : Bool;   // Manueller Ansteuerbefehl für Grundstellung
      actor : "typeActor";
      signals : "typeStationSignals";
      manualMovement : "typeManualMovements";
   END_VAR
   VAR
      statManualMovementNo : UInt;
      statStationNo : USInt;
      statMoveNoInStation : UInt;
   END_VAR
   VAR_TEMP
      tempInitialised : Bool;
      tempRelease : Bool;
   END_VAR
   VAR_TEMP   // added for the SCL form of the ladder/FBD networks
      _w1 : Bool;
   END_VAR
BEGIN

REGION Network 1: Initialisierungsprozess für eine Einrichtfunktion
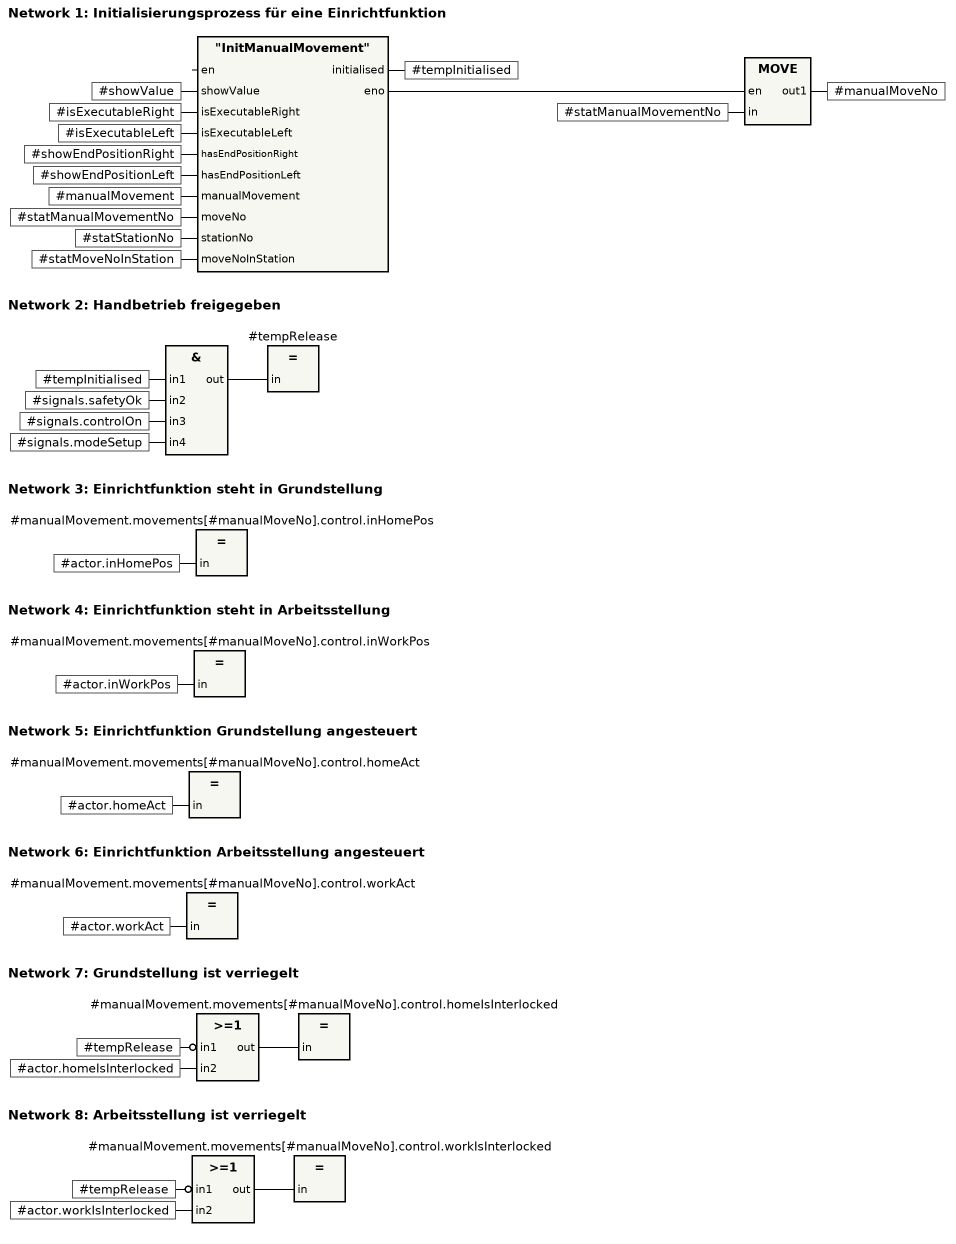
   "InitManualMovement"(showValue := #showValue,
                        isExecutableRight := #isExecutableRight,
                        isExecutableLeft := #isExecutableLeft,
                        hasEndPositionRight := #showEndPositionRight,
                        hasEndPositionLeft := #showEndPositionLeft,
                        manualMovement := #manualMovement,
                        moveNo := #statManualMovementNo,
                        stationNo := #statStationNo,
                        moveNoInStation := #statMoveNoInStation,
                        initialised => #tempInitialised,
                        ENO => #_w1);
   IF #_w1 THEN #manualMoveNo := #statManualMovementNo; END_IF;
END_REGION

REGION Network 2: Handbetrieb freigegeben
   #tempRelease := #tempInitialised AND #signals.safetyOk AND #signals.controlOn AND #signals.modeSetup;
END_REGION

REGION Network 3: Einrichtfunktion steht in Grundstellung
   #manualMovement.movements[#manualMoveNo].control.inHomePos := #actor.inHomePos;
END_REGION

REGION Network 4: Einrichtfunktion steht in Arbeitsstellung
   #manualMovement.movements[#manualMoveNo].control.inWorkPos := #actor.inWorkPos;
END_REGION

REGION Network 5: Einrichtfunktion Grundstellung angesteuert
   #manualMovement.movements[#manualMoveNo].control.homeAct := #actor.homeAct;
END_REGION

REGION Network 6: Einrichtfunktion Arbeitsstellung angesteuert
   #manualMovement.movements[#manualMoveNo].control.workAct := #actor.workAct;
END_REGION

REGION Network 7: Grundstellung ist verriegelt
   #manualMovement.movements[#manualMoveNo].control.homeIsInterlocked := NOT #tempRelease OR #actor.homeIsInterlocked;
END_REGION

REGION Network 8: Arbeitsstellung ist verriegelt
   #manualMovement.movements[#manualMoveNo].control.workIsInterlocked := NOT #tempRelease OR #actor.workIsInterlocked;
END_REGION

REGION Network 9: Rücksetze manuelle Bewegungsansteuerung des Aktors
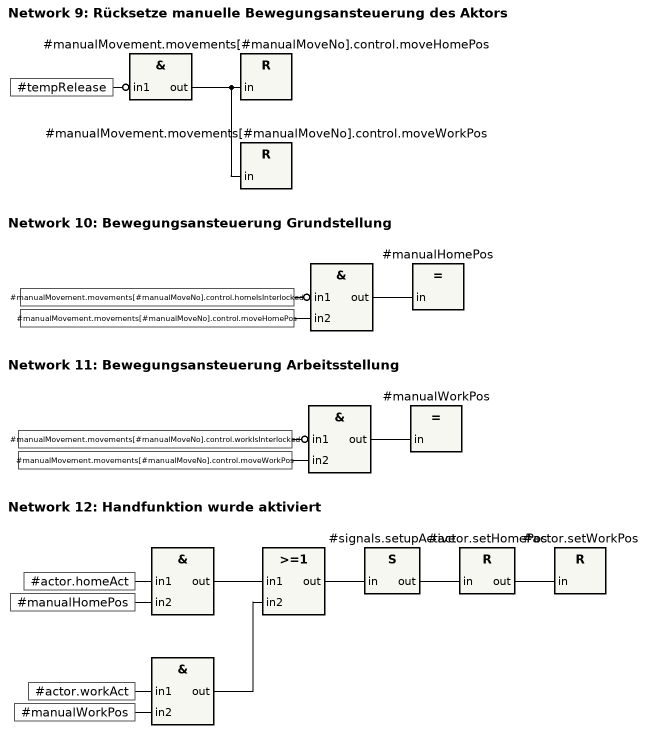
   IF NOT #tempRelease THEN
       #manualMovement.movements[#manualMoveNo].control.moveHomePos := FALSE;
       #manualMovement.movements[#manualMoveNo].control.moveWorkPos := FALSE;
   END_IF;
END_REGION

REGION Network 10: Bewegungsansteuerung Grundstellung
   #manualHomePos := NOT #manualMovement.movements[#manualMoveNo].control.homeIsInterlocked AND #manualMovement.movements[#manualMoveNo].control.moveHomePos;
END_REGION

REGION Network 11: Bewegungsansteuerung Arbeitsstellung
   #manualWorkPos := NOT #manualMovement.movements[#manualMoveNo].control.workIsInterlocked AND #manualMovement.movements[#manualMoveNo].control.moveWorkPos;
END_REGION

REGION Network 12: Handfunktion wurde aktiviert
   IF (#actor.homeAct AND #manualHomePos) OR (#actor.workAct AND #manualWorkPos) THEN
       #signals.setupActive := TRUE;
       #actor.setHomePos := FALSE;
       #actor.setWorkPos := FALSE;
   END_IF;
END_REGION
END_FUNCTION_BLOCK

FUNCTION_BLOCK "DriveManualMovementJog"   // FB910, FBD
TITLE = Einrichtfunktion Tippen für einen Servo
{ S7_Optimized_Access := 'TRUE' }
VERSION : 0.1
// Ersteller: Andreas Fast Automation
// E-Mail: automation@fast-andreas.de
// 
// Projekt dient zu Demonstrationszwecken und frei genutzt werden.
// 
// Bausteinbeschreibung:
   VAR_INPUT
      status : "typeDriveStatus";   // Status
   END_VAR
   VAR_OUTPUT
      manualMoveNo : UInt;
   END_VAR
   VAR_IN_OUT
      control : "typeDriveControl";   // Steuerbefehle
      signals : "typeStationSignals";
      manualMovement : "typeManualMovements";
   END_VAR
   VAR
      statActor : "typeActor";
      instActorManualMovement : "ActorManualMovement";
   END_VAR
   VAR_TEMP
      tempInitialised : Bool;
      tempRelease : Bool;
   END_VAR
BEGIN

REGION Network 1: steht in Grundstellung
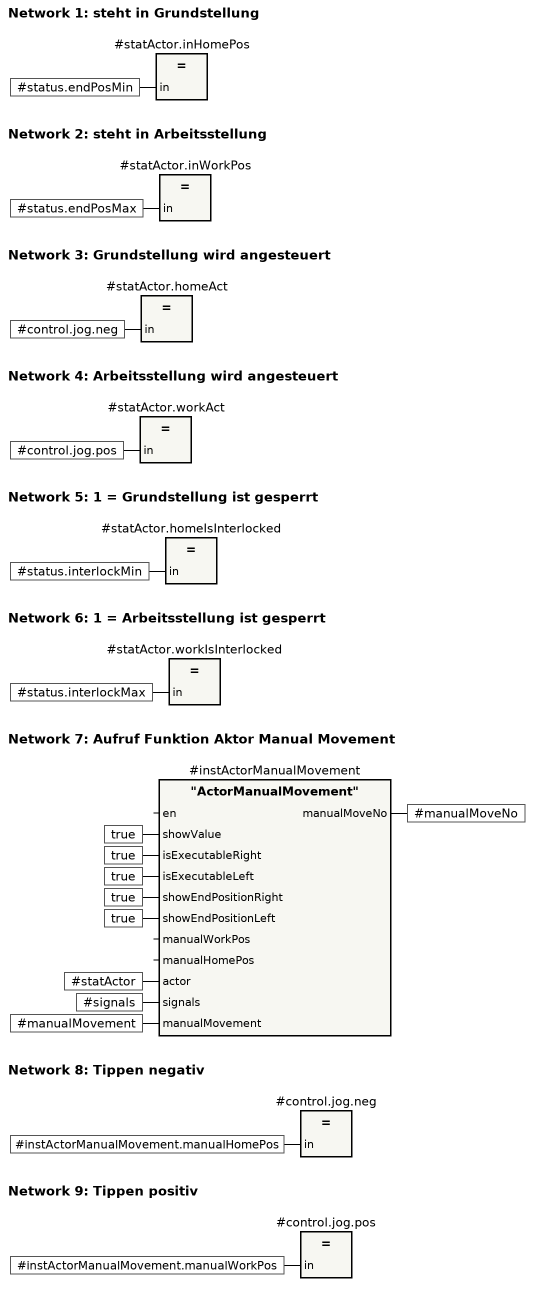
   #statActor.inHomePos := #status.endPosMin;
END_REGION

REGION Network 2: steht in Arbeitsstellung
   #statActor.inWorkPos := #status.endPosMax;
END_REGION

REGION Network 3: Grundstellung wird angesteuert
   #statActor.homeAct := #control.jog.neg;
END_REGION

REGION Network 4: Arbeitsstellung wird angesteuert
   #statActor.workAct := #control.jog.pos;
END_REGION

REGION Network 5: 1 = Grundstellung ist gesperrt
   #statActor.homeIsInterlocked := #status.interlockMin;
END_REGION

REGION Network 6: 1 = Arbeitsstellung ist gesperrt
   #statActor.workIsInterlocked := #status.interlockMax;
END_REGION

REGION Network 7: Aufruf Funktion Aktor Manual Movement
   #instActorManualMovement(showValue := true,   // "ActorManualMovement"
                           isExecutableRight := true,
                           isExecutableLeft := true,
                           showEndPositionRight := true,
                           showEndPositionLeft := true,
                           actor := #statActor,
                           signals := #signals,
                           manualMovement := #manualMovement,
                           manualMoveNo => #manualMoveNo);
END_REGION

REGION Network 8: Tippen negativ
   #control.jog.neg := #instActorManualMovement.manualHomePos;
END_REGION

REGION Network 9: Tippen positiv
   #control.jog.pos := #instActorManualMovement.manualWorkPos;
END_REGION

REGION Network 10: Istposition in Einrichtfunktion anzeigen
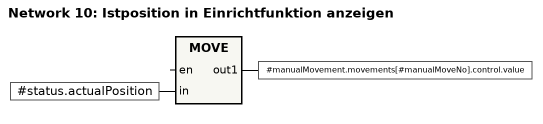
   #manualMovement.movements[#manualMoveNo].control.value := #status.actualPosition;
END_REGION
END_FUNCTION_BLOCK

FUNCTION "InitManualMovement" : Void   // FC907, FBD
TITLE = Initialisierungsprozess für eine Einrichtfunktion
{ S7_Optimized_Access := 'TRUE' }
VERSION : 0.1
// Ersteller: Andreas Fast Automation
// E-Mail: automation@fast-andreas.de
// 
// Projekt dient zu Demonstrationszwecken und frei genutzt werden.
// 
// Bausteinbeschreibung:
   VAR_INPUT
      showValue : Bool;   // Zeige Dezimalanzeige
      isExecutableRight : Bool;   // Ist ausführbar rechte Seite
      isExecutableLeft : Bool;   // Ist ausführbar linke Seite
      hasEndPositionRight : Bool;   // Zeige Endposition rechte Seite
      hasEndPositionLeft : Bool;   // Zeige Endposition linke Seite
   END_VAR
   VAR_OUTPUT
      initialised : Bool;
   END_VAR
   VAR_IN_OUT
      manualMovement : "typeManualMovements";
      moveNo : UInt;
      stationNo : USInt;
      moveNoInStation : UInt;
   END_VAR
   VAR_TEMP   // added for the SCL form of the ladder/FBD networks
      _w1 : Bool;
   END_VAR
BEGIN

REGION Network 1: Plausibilitätsprüfung/Initialisierung läuft
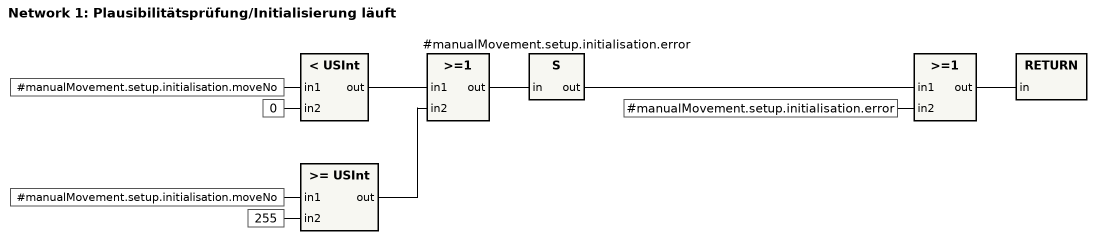
   #_w1 := (#manualMovement.setup.initialisation.moveNo < 0) OR (#manualMovement.setup.initialisation.moveNo >= 255);
   IF #_w1 THEN #manualMovement.setup.initialisation.error := TRUE; END_IF;
   IF #_w1 OR #manualMovement.setup.initialisation.error THEN
       ENO := TRUE;
       RETURN;
   END_IF;
END_REGION

REGION Network 2: Initialisierung
